KUKA KRL program: MyProgram_085().src

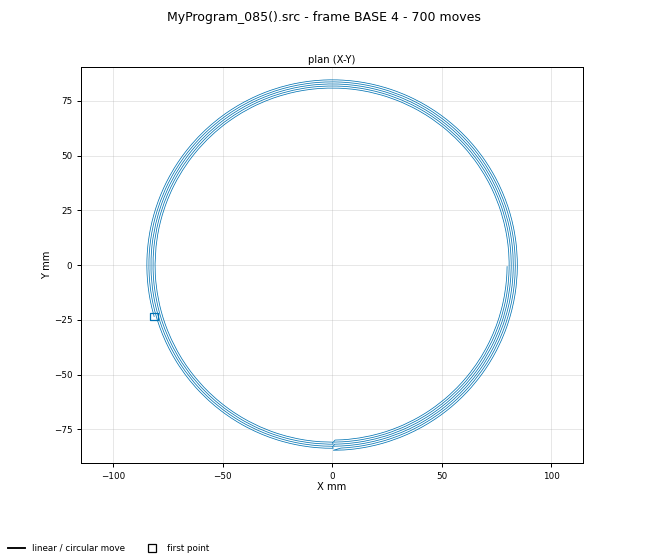
[picture p0: tool path of MyProgram_085().src in frame BASE 4, 700 of 700 moves have a stored position in this frame; points joined in program order, loops and branches not executed]
&ACCESS RVP
&REL 1
&PARAM TEMPLATE = C:\KRC\Roboter\Template\vorgabe
&PARAM EDITMASK = *
DEF MyProgram_085()
; ---- Setting reference (Base) ----
$BASE = BASE_DATA[4]

; --------------------------
; ---- Setting tool (TCP) ----
$TOOL = TOOL_DATA[3]
; --------------------------

$VEL.CP = VEL_APROX_PRINT
Startdeposition()
$VEL.CP = VEL_PRINT
LIN {X -81.258,Y -23.4932,Z 84,A -170.2717,B 24.9188,C -2.0806,E1 24.845,E2 255.2364} C_DIS
LIN {X -82.3528,Y -19.3072,Z 84,A -172.0172,B 24.9156,C -2.1214,E1 24.8439,E2 256.895} C_DIS
LIN {X -83.0894,Y -15.8383,Z 84,A -174.5177,B 24.9152,C -2.1261,E1 24.8425,E2 259.3989} C_DIS
LIN {X -83.5159,Y -13.4174,Z 84,A -176.5241,B 24.9155,C -2.122,E1 24.8416,E2 261.4269} C_DIS
LIN {X -83.9859,Y -10.0545,Z 84,A -178.7567,B 24.9148,C -2.1311,E1 24.8408,E2 263.6513} C_DIS
LIN {X -84.2675,Y -7.3389,Z 84,A 179.2872,B 24.9146,C -2.134,E1 24.8402,E2 265.6121} C_DIS
LIN {X -84.4963,Y -3.8886,Z 84,A 177.017,B 24.9138,C -2.1434,E1 24.8399,E2 267.8736} C_DIS
LIN {X -84.5836,Y -0.541,Z 84,A 174.7604,B 24.9132,C -2.1509,E1 24.8398,E2 270.1257} C_DIS
LIN {X -84.5494,Y 2.4664,Z 84,A 172.6653,B 24.9128,C -2.1559,E1 24.8399,E2 272.2217} C_DIS
LIN {X -84.435,Y 5.055,Z 84,A 170.8313,B 24.9125,C -2.1594,E1 24.8402,E2 274.0584} C_DIS
LIN {X -84.1499,Y 8.5742,Z 84,A 168.4952,B 24.9118,C -2.1685,E1 24.8408,E2 276.3867} C_DIS
LIN {X -83.8432,Y 11.1849,Z 84,A 166.6416,B 24.9115,C -2.1722,E1 24.8414,E2 278.2425} C_DIS
LIN {X -83.3207,Y 14.5775,Z 84,A 164.375,B 24.9108,C -2.1812,E1 24.8424,E2 280.5012} C_DIS
LIN {X -82.9257,Y 16.6767,Z 84,A 162.9181,B 24.9104,C -2.1855,E1 24.8432,E2 281.9565} C_DIS
LIN {X -82.2344,Y 19.8053,Z 84,A 160.6347,B 24.9101,C -2.1893,E1 24.8447,E2 284.2441} C_DIS
LIN {X -81.3682,Y 23.1062,Z 84,A 158.4682,B 24.9092,C -2.2004,E1 24.8463,E2 286.3966} C_DIS
LIN {X -80.4587,Y 26.0974,Z 84,A 156.0154,B 24.9094,C -2.198,E1 24.8483,E2 288.8692} C_DIS
LIN {X -79.338,Y 29.3307,Z 84,A 153.7423,B 24.9087,C -2.2063,E1 24.8505,E2 291.1354} C_DIS
LIN {X -78.306,Y 31.9821,Z 84,A 151.9175,B 24.908,C -2.2149,E1 24.8524,E2 292.9499} C_DIS
LIN {X -76.9778,Y 35.06,Z 84,A 149.7082,B 24.9073,C -2.2233,E1 24.8549,E2 295.1512} C_DIS
LIN {X -75.657,Y 37.8257,Z 84,A 147.6321,B 24.9068,C -2.2295,E1 24.8574,E2 297.2238} C_DIS
LIN {X -74.2269,Y 40.56,Z 84,A 145.2417,B 24.9069,C -2.2275,E1 24.8606,E2 299.6317} C_DIS
LIN {X -72.1363,Y 44.1714,Z 84,A 142.1378,B 24.9069,C -2.228,E1 24.8651,E2 302.7503} C_DIS
LIN {X -70.3586,Y 46.9528,Z 84,A 140.6207,B 24.9047,C -2.2536,E1 24.8673,E2 304.2139} C_DIS
LIN {X -68.1618,Y 50.0866,Z 84,A 137.8462,B 24.9045,C -2.2557,E1 24.8718,E2 306.997} C_DIS
LIN {X -66.2766,Y 52.5558,Z 84,A 135.0425,B 24.9057,C -2.2423,E1 24.8767,E2 309.8459} C_DIS
LIN {X -63.9412,Y 55.3742,Z 84,A 133.1912,B 24.9037,C -2.2657,E1 24.88,E2 311.6499} C_DIS
LIN {X -61.115,Y 58.4779,Z 84,A 130.1814,B 24.9035,C -2.2681,E1 24.8858,E2 314.667} C_DIS
LIN {X -58.0046,Y 61.5642,Z 84,A 127.0353,B 24.9033,C -2.2703,E1 24.8921,E2 317.8211} C_DIS
LIN {X -55.2393,Y 64.0587,Z 84,A 124.5405,B 24.9028,C -2.2767,E1 24.8973,E2 320.3105} C_DIS
LIN {X -51.7634,Y 66.8974,Z 84,A 121.7058,B 24.9017,C -2.2889,E1 24.9035,E2 323.1267} C_DIS
LIN {X -48.6455,Y 69.1989,Z 84,A 119.0158,B 24.9014,C -2.2924,E1 24.9096,E2 325.8177} C_DIS
LIN {X -46.1517,Y 70.8868,Z 84,A 116.9277,B 24.9012,C -2.2949,E1 24.9144,E2 327.9066} C_DIS
LIN {X -42.9543,Y 72.8671,Z 84,A 114.5021,B 24.9005,C -2.303,E1 24.9202,E2 330.3205} C_DIS
LIN {X -39.9938,Y 74.534,Z 84,A 111.9144,B 24.9008,C -2.2989,E1 24.9266,E2 332.9254} C_DIS
LIN {X -36.3147,Y 76.394,Z 84,A 109.3731,B 24.8999,C -2.3104,E1 24.9329,E2 335.4459} C_DIS
LIN {X -33.3203,Y 77.747,Z 84,A 107.1231,B 24.8996,C -2.3129,E1 24.9386,E2 337.6952} C_DIS
LIN {X -30.5085,Y 78.8929,Z 84,A 105.0579,B 24.8994,C -2.3155,E1 24.944,E2 339.7588} C_DIS
LIN {X -27.9226,Y 79.8437,Z 84,A 103.2111,B 24.8992,C -2.3184,E1 24.9489,E2 341.6024} C_DIS
LIN {X -23.5033,Y 81.2557,Z 84,A 99.7544,B 24.8996,C -2.3129,E1 24.9581,E2 345.0781} C_DIS
LIN {X -19.3603,Y 82.3405,Z 84,A 97.4785,B 24.8978,C -2.3338,E1 24.9642,E2 347.3076} C_DIS
LIN {X -17.0374,Y 82.8517,Z 84,A 95.5853,B 24.8984,C -2.3269,E1 24.9694,E2 349.2193} C_DIS
LIN {X -14.0779,Y 83.4057,Z 84,A 93.6062,B 24.8981,C -2.3302,E1 24.9748,E2 351.1926} C_DIS
LIN {X -10.9036,Y 83.8796,Z 84,A 91.394,B 24.8981,C -2.3305,E1 24.9809,E2 353.4059} C_DIS
LIN {X -7.5623,Y 84.2469,Z 84,A 88.9914,B 24.8983,C -2.328,E1 24.9876,E2 355.8159} C_DIS
LIN {X -3.933,Y 84.4944,Z 84,A 86.7832,B 24.8976,C -2.3365,E1 24.9937,E2 358.0046} C_DIS
LIN {X -1.2539,Y 84.5766,Z 84,A 84.7108,B 24.8982,C -2.3293,E1 24.9996,E2 360.0941} C_DIS
LIN {X 2.2908,Y 84.5548,Z 84,A 82.3368,B 24.8981,C -2.3305,E1 25.0062,E2 362.4651} C_DIS
LIN {X 4.9822,Y 84.439,Z 84,A 80.504,B 24.8981,C -2.3303,E1 25.0113,E2 364.2977} C_DIS
LIN {X 8.2772,Y 84.1808,Z 84,A 78.427,B 24.8977,C -2.3349,E1 25.017,E2 366.3625} C_DIS
LIN {X 11.0872,Y 83.8558,Z 84,A 76.403,B 24.898,C -2.3313,E1 25.0227,E2 368.3934} C_DIS
LIN {X 14.4147,Y 83.3494,Z 84,A 74.0384,B 24.8983,C -2.328,E1 25.0292,E2 370.7636} C_DIS
LIN {X 17.8759,Y 82.675,Z 84,A 71.6875,B 24.8983,C -2.3281,E1 25.0356,E2 373.1113} C_DIS
LIN {X 21.1707,Y 81.8932,Z 84,A 69.4403,B 24.8983,C -2.3282,E1 25.0417,E2 375.355} C_DIS
LIN {X 24.6364,Y 80.9192,Z 84,A 67.2437,B 24.8978,C -2.3339,E1 25.0476,E2 377.5343} C_DIS
LIN {X 26.9465,Y 80.1784,Z 84,A 65.4111,B 24.8984,C -2.3268,E1 25.0524,E2 379.3803} C_DIS
LIN {X 29.6504,Y 79.2189,Z 84,A 62.8102,B 24.9003,C -2.3047,E1 25.0594,E2 382.028} C_DIS
LIN {X 32.942,Y 77.9071,Z 84,A 61.3092,B 24.8981,C -2.3301,E1 25.0631,E2 383.4654} C_DIS
LIN {X 35.0479,Y 76.9832,Z 84,A 59.6938,B 24.8984,C -2.3265,E1 25.0672,E2 385.0853} C_DIS
LIN {X 37.4119,Y 75.862,Z 84,A 57.6987,B 24.8992,C -2.3174,E1 25.0723,E2 387.0968} C_DIS
LIN {X 40.5488,Y 74.2329,Z 84,A 55.247,B 24.8997,C -2.3124,E1 25.0783,E2 389.5533} C_DIS
LIN {X 43.6284,Y 72.4663,Z 84,A 52.8273,B 24.9,C -2.3085,E1 25.0842,E2 391.9749} C_DIS
LIN {X 46.9407,Y 70.3665,Z 84,A 50.2167,B 24.9003,C -2.3058,E1 25.0903,E2 394.5835} C_DIS
LIN {X 49.6746,Y 68.4634,Z 84,A 48.0134,B 24.9004,C -2.3037,E1 25.0953,E2 396.7841} C_DIS
LIN {X 52.2744,Y 66.4989,Z 84,A 45.8438,B 24.9007,C -2.3009,E1 25.1001,E2 398.9522} C_DIS
LIN {X 54.843,Y 64.3966,Z 84,A 43.7202,B 24.9007,C -2.3007,E1 25.1046,E2 401.0682} C_DIS
LIN {X 56.9564,Y 62.5359,Z 84,A 41.8463,B 24.9009,C -2.298,E1 25.1085,E2 402.941} C_DIS
LIN {X 59.0852,Y 60.5299,Z 84,A 39.6486,B 24.9019,C -2.2869,E1 25.113,E2 405.1558} C_DIS
LIN {X 61.4852,Y 58.0886,Z 84,A 37.4909,B 24.9019,C -2.2871,E1 25.1172,E2 407.3036} C_DIS
LIN {X 64.1932,Y 55.0818,Z 84,A 34.6835,B 24.9026,C -2.2788,E1 25.1224,E2 410.1182} C_DIS
LIN {X 66.2537,Y 52.5847,Z 84,A 32.5055,B 24.903,C -2.2741,E1 25.1262,E2 412.2971} C_DIS
LIN {X 68.4835,Y 49.6473,Z 84,A 30.195,B 24.903,C -2.2741,E1 25.13,E2 414.5964} C_DIS
LIN {X 70.0955,Y 47.3425,Z 84,A 28.0798,B 24.904,C -2.2625,E1 25.1334,E2 416.7288} C_DIS
LIN {X 71.8637,Y 44.6132,Z 84,A 25.9695,B 24.9042,C -2.2599,E1 25.1366,E2 418.8348} C_DIS
LIN {X 73.3555,Y 42.1147,Z 84,A 24.0489,B 24.9045,C -2.2563,E1 25.1393,E2 420.7539} C_DIS
LIN {X 74.5437,Y 39.976,Z 84,A 22.2403,B 24.9053,C -2.2468,E1 25.1417,E2 422.5754} C_DIS
LIN {X 76.1666,Y 36.7879,Z 84,A 19.9576,B 24.9055,C -2.2448,E1 25.1445,E2 424.8508} C_DIS
LIN {X 77.7532,Y 33.3037,Z 84,A 16.6318,B 24.9081,C -2.2133,E1 25.1483,E2 428.2328} C_DIS
LIN {X 79.201,Y 29.6977,Z 84,A 14.5929,B 24.9071,C -2.2252,E1 25.1503,E2 430.2322} C_DIS
LIN {X 80.3308,Y 26.4926,Z 84,A 12.4263,B 24.9073,C -2.2228,E1 25.1522,E2 432.3922} C_DIS
LIN {X 81.2016,Y 23.6879,Z 84,A 10.4534,B 24.9078,C -2.2174,E1 25.1538,E2 434.3665} C_DIS
LIN {X 82.0478,Y 20.569,Z 84,A 8.2194,B 24.9084,C -2.2093,E1 25.1554,E2 436.6069} C_DIS
LIN {X 82.8109,Y 17.2361,Z 84,A 5.9479,B 24.9089,C -2.2037,E1 25.1568,E2 438.8784} C_DIS
LIN {X 83.338,Y 14.4812,Z 84,A 4.0007,B 24.9095,C -2.1962,E1 25.1577,E2 440.832} C_DIS
LIN {X 83.8789,Y 10.9088,Z 84,A 1.8383,B 24.9094,C -2.1981,E1 25.1586,E2 442.9771} C_DIS
LIN {X 84.2078,Y 7.9856,Z 84,A -0.6462,B 24.9112,C -2.1753,E1 25.1593,E2 445.5006} C_DIS
LIN {X 84.5468,Y 2.554,Z 84,A -4.3801,B 24.9123,C -2.162,E1 25.1598,E2 449.2437} C_DIS
LIN {X 84.5806,Y -1.0264,Z 84,A -6.4606,B 24.912,C -2.1658,E1 25.1598,E2 451.303} C_DIS
LIN {X 84.4797,Y -4.247,Z 84,A -8.5268,B 24.9123,C -2.1627,E1 25.1595,E2 453.3642} C_DIS
LIN {X 83.9739,Y -10.1565,Z 84,A -12.6253,B 24.9135,C -2.1471,E1 25.1584,E2 457.4751} C_DIS
LIN {X 83.5288,Y -13.3334,Z 84,A -15.2054,B 24.9152,C -2.1266,E1 25.1573,E2 460.0886} C_DIS
LIN {X 82.9598,Y -16.5061,Z 84,A -17.3336,B 24.9156,C -2.1215,E1 25.1561,E2 462.2163} C_DIS
LIN {X 82.0892,Y -20.4002,Z 84,A -19.606,B 24.9151,C -2.1273,E1 25.1547,E2 464.4618} C_DIS
LIN {X 81.2074,Y -23.6685,Z 84,A -21.9819,B 24.9159,C -2.1174,E1 25.1529,E2 466.8476} C_DIS
LIN {X 80.088,Y -27.2145,Z 84,A -24.189,B 24.9157,C -2.12,E1 25.151,E2 469.0359} C_DIS
LIN {X 78.9874,Y -30.2617,Z 84,A -26.4098,B 24.9163,C -2.1124,E1 25.1488,E2 471.2624} C_DIS
LIN {X 77.352,Y -34.2281,Z 84,A -30.4851,B 24.9201,C -2.0648,E1 25.1442,E2 475.4278} C_DIS
LIN {X 75.1596,Y -38.8052,Z 84,A -32.3854,B 24.9168,C -2.1057,E1 25.142,E2 477.2213} C_DIS
LIN {X 73.4267,Y -41.9908,Z 84,A -35.7576,B 24.9198,C -2.068,E1 25.1373,E2 480.6649} C_DIS
LIN {X 71.7723,Y -44.7595,Z 84,A -37.2898,B 24.9186,C -2.0835,E1 25.1351,E2 482.1527} C_DIS
LIN {X 70.1825,Y -47.214,Z 84,A -39.3837,B 24.9193,C -2.0742,E1 25.1319,E2 484.2582} C_DIS
LIN {X 68.3451,Y -49.8363,Z 84,A -41.5585,B 24.9198,C -2.0681,E1 25.1283,E2 486.4368} C_DIS
LIN {X 66.5336,Y -52.2306,Z 84,A -43.9673,B 24.9212,C -2.0503,E1 25.1242,E2 488.8764} C_DIS
LIN {X 63.5973,Y -55.7682,Z 84,A -46.5786,B 24.9205,C -2.0589,E1 25.1195,E2 491.4554} C_DIS
LIN {X 61.6049,Y -57.9613,Z 84,A -48.5956,B 24.9209,C -2.0535,E1 25.1157,E2 493.4762} C_DIS
LIN {X 59.4587,Y -60.161,Z 84,A -50.6632,B 24.9213,C -2.0489,E1 25.1116,E2 495.546} C_DIS
LIN {X 57.2741,Y -62.2444,Z 84,A -52.8275,B 24.9219,C -2.0402,E1 25.1072,E2 497.722} C_DIS
LIN {X 54.4849,Y -64.7017,Z 84,A -55.2672,B 24.9222,C -2.037,E1 25.102,E2 500.1595} C_DIS
LIN {X 52.1024,Y -66.6349,Z 84,A -57.3582,B 24.9226,C -2.0321,E1 25.0974,E2 502.2544} C_DIS
LIN {X 49.6131,Y -68.5085,Z 84,A -59.3441,B 24.9226,C -2.0318,E1 25.093,E2 504.234} C_DIS
LIN {X 46.7155,Y -70.5151,Z 84,A -61.7837,B 24.9231,C -2.0254,E1 25.0873,E2 506.6805} C_DIS
LIN {X 44.0739,Y -72.1955,Z 84,A -63.9286,B 24.9234,C -2.0206,E1 25.0822,E2 508.8298} C_DIS
LIN {X 40.9406,Y -74.0179,Z 84,A -67.0141,B 24.9253,C -1.996,E1 25.0746,E2 511.9643} C_DIS
LIN {X 37.734,Y -75.7024,Z 84,A -68.9066,B 24.9243,C -2.0099,E1 25.07,E2 513.8188} C_DIS
LIN {X 34.381,Y -77.2838,Z 84,A -71.9632,B 24.9258,C -1.9887,E1 25.0621,E2 516.9181} C_DIS
LIN {X 31.0532,Y -78.6791,Z 84,A -73.3423,B 24.9236,C -2.0192,E1 25.0587,E2 518.2219} C_DIS
LIN {X 25.9181,Y -80.5167,Z 84,A -77.3653,B 24.9247,C -2.0039,E1 25.0481,E2 522.2728} C_DIS
LIN {X 23.0747,Y -81.3771,Z 84,A -79.3426,B 24.9247,C -2.0028,E1 25.0428,E2 524.2494} C_DIS
LIN {X 20.0403,Y -82.177,Z 84,A -81.8961,B 24.926,C -1.9872,E1 25.0358,E2 526.836} C_DIS
LIN {X 16.4441,Y -82.9728,Z 84,A -83.8435,B 24.9248,C -2.0021,E1 25.0306,E2 528.7456} C_DIS
LIN {X 13.908,Y -83.4341,Z 84,A -85.8616,B 24.9256,C -1.9923,E1 25.0249,E2 530.7849} C_DIS
LIN {X 10.3473,Y -83.9514,Z 84,A -88.0451,B 24.9251,C -1.9985,E1 25.0189,E2 532.9517} C_DIS
LIN {X 7.3763,Y -84.264,Z 84,A -90.0792,B 24.9252,C -1.9971,E1 25.0133,E2 534.9878} C_DIS
LIN {X 5.3469,Y -84.4169,Z 84,A -91.6987,B 24.9258,C -1.989,E1 25.0087,E2 536.6258} C_DIS
LIN {X 0.5554,Y -84.5445,Z 84,A -94.0902,B 24.9239,C -2.0151,E1 25.0023,E2 538.9549} C_DIS
Enddeposition()
LIN {X 0.5554,Y -84.5445,Z 84,A -94.0902,B 24.9239,C -2.0151,E1 25.0023,E2 538.9549} C_DIS
Startdeposition()
$VEL.CP = VEL_PRINT
LIN {X 4.0199,Y -83.5536,Z 84,A -91.4821,B 24.9221,C -2.0387,E1 25.0097,E2 536.2916} C_DIS
LIN {X 7.177,Y -83.3423,Z 84,A -88.8971,B 24.921,C -2.0528,E1 25.0169,E2 533.6745} C_DIS
LIN {X 11.2811,Y -82.8861,Z 84,A -86.5387,B 24.922,C -2.0398,E1 25.0234,E2 531.3487} C_DIS
LIN {X 14.1672,Y -82.4416,Z 84,A -84.4181,B 24.9216,C -2.0451,E1 25.0293,E2 529.2177} C_DIS
LIN {X 18.2064,Y -81.6443,Z 84,A -81.4549,B 24.921,C -2.0521,E1 25.0374,E2 526.2417} C_DIS
LIN {X 23.7052,Y -80.22,Z 84,A -77.9146,B 24.9216,C -2.0451,E1 25.0469,E2 522.7236} C_DIS
LIN {X 26.3192,Y -79.4006,Z 84,A -75.1328,B 24.9191,C -2.0764,E1 25.0544,E2 519.8729} C_DIS
LIN {X 30.3174,Y -77.9623,Z 84,A -73.2321,B 24.9214,C -2.0478,E1 25.0592,E2 518.0441} C_DIS
LIN {X 34.0465,Y -76.4077,Z 84,A -70.3229,B 24.9207,C -2.0564,E1 25.0667,E2 515.1215} C_DIS
LIN {X 35.9853,Y -75.5137,Z 84,A -68.6164,B 24.9199,C -2.0666,E1 25.0711,E2 513.3953} C_DIS
LIN {X 40.6616,Y -73.1016,Z 84,A -65.0227,B 24.9195,C -2.0724,E1 25.0799,E2 509.7981} C_DIS
LIN {X 45.2214,Y -70.3719,Z 84,A -60.7698,B 24.9173,C -2.0994,E1 25.0901,E2 505.4948} C_DIS
LIN {X 48.8035,Y -67.9373,Z 84,A -58.3698,B 24.9183,C -2.0867,E1 25.0955,E2 503.1333} C_DIS
LIN {X 52.051,Y -65.4823,Z 84,A -55.9631,B 24.9189,C -2.0801,E1 25.1007,E2 500.7511} C_DIS
LIN {X 54.2015,Y -63.7133,Z 84,A -54.2455,B 24.919,C -2.0781,E1 25.1044,E2 499.0447} C_DIS
LIN {X 57.1138,Y -61.1168,Z 84,A -50.9148,B 24.9168,C -2.1061,E1 25.1114,E2 495.6614} C_DIS
LIN {X 60.324,Y -57.9501,Z 84,A -48.2074,B 24.9172,C -2.1009,E1 25.1166,E2 492.9778} C_DIS
LIN {X 62.4733,Y -55.6266,Z 84,A -45.5471,B 24.9155,C -2.1228,E1 25.1217,E2 490.2776} C_DIS
LIN {X 64.6916,Y -53.031,Z 84,A -43.7656,B 24.9165,C -2.1102,E1 25.1248,E2 488.534} C_DIS
LIN {X 68.6131,Y -47.8481,Z 84,A -38.7416,B 24.914,C -2.1415,E1 25.1331,E2 483.4604} C_DIS
LIN {X 70.6127,Y -44.8463,Z 84,A -36.3085,B 24.9135,C -2.1472,E1 25.1368,E2 481.0261} C_DIS
LIN {X 72.409,Y -41.8828,Z 84,A -34.6666,B 24.915,C -2.1293,E1 25.139,E2 479.4348} C_DIS
LIN {X 74.0802,Y -38.8501,Z 84,A -32.4822,B 24.915,C -2.1299,E1 25.1419,E2 477.2604} C_DIS
LIN {X 76.2889,Y -34.3102,Z 84,A -28.9902,B 24.914,C -2.1413,E1 25.1462,E2 473.7603} C_DIS
LIN {X 77.8847,Y -30.515,Z 84,A -25.8854,B 24.9125,C -2.1594,E1 25.1495,E2 470.6298} C_DIS
LIN {X 79.1087,Y -27.1888,Z 84,A -22.8184,B 24.9101,C -2.1886,E1 25.1523,E2 467.5111} C_DIS
LIN {X 80.2758,Y -23.5171,Z 84,A -20.9909,B 24.9117,C -2.1693,E1 25.1538,E2 465.7397} C_DIS
LIN {X 81.0511,Y -20.6864,Z 84,A -19.0499,B 24.9114,C -2.1733,E1 25.1551,E2 463.8005} C_DIS
LIN {X 81.9401,Y -16.8226,Z 84,A -15.9084,B 24.9095,C -2.1963,E1 25.157,E2 460.6229} C_DIS
LIN {X 82.6235,Y -13.0619,Z 84,A -13.2409,B 24.9087,C -2.2063,E1 25.1582,E2 457.9474} C_DIS
LIN {X 83.0754,Y -9.7807,Z 84,A -10.9669,B 24.9081,C -2.2137,E1 25.159,E2 455.6693} C_DIS
LIN {X 83.4824,Y -5.2907,Z 84,A -7.8895,B 24.9073,C -2.2232,E1 25.1596,E2 452.5877} C_DIS
LIN {X 83.6471,Y -0.6032,Z 84,A -3.9008,B 24.9042,C -2.2601,E1 25.1597,E2 448.5358} C_DIS
LIN {X 83.5087,Y 4.8515,Z 84,A -1.6888,B 24.9076,C -2.22,E1 25.1595,E2 446.4316} C_DIS
LIN {X 83.3102,Y 7.5248,Z 84,A 0.3928,B 24.9064,C -2.2341,E1 25.159,E2 444.3291} C_DIS
LIN {X 82.9542,Y 10.7605,Z 84,A 2.5084,B 24.9061,C -2.2372,E1 25.1583,E2 442.2185} C_DIS
LIN {X 82.5337,Y 13.6166,Z 84,A 4.5625,B 24.9054,C -2.246,E1 25.1574,E2 440.1558} C_DIS
LIN {X 81.966,Y 16.6967,Z 84,A 6.6673,B 24.9049,C -2.2513,E1 25.1563,E2 438.0509} C_DIS
LIN {X 81.2888,Y 19.7312,Z 84,A 8.4277,B 24.9054,C -2.2454,E1 25.1552,E2 436.3145} C_DIS
LIN {X 80.2379,Y 23.6451,Z 84,A 11.5985,B 24.9036,C -2.267,E1 25.1529,E2 433.111} C_DIS
LIN {X 79.2298,Y 26.8297,Z 84,A 14.4891,B 24.9013,C -2.294,E1 25.1502,E2 430.1728} C_DIS
LIN {X 78.0075,Y 30.202,Z 84,A 16.0399,B 24.9033,C -2.2708,E1 25.1488,E2 428.6856} C_DIS
LIN {X 76.2468,Y 34.4035,Z 84,A 19.2998,B 24.9021,C -2.2843,E1 25.1452,E2 425.4115} C_DIS
LIN {X 75.0446,Y 36.9533,Z 84,A 21.295,B 24.9015,C -2.2918,E1 25.1428,E2 423.4093} C_DIS
LIN {X 73.6627,Y 39.6367,Z 84,A 23.3793,B 24.9009,C -2.298,E1 25.14,E2 421.3214} C_DIS
LIN {X 72.552,Y 41.634,Z 84,A 25.2545,B 24.8997,C -2.3125,E1 25.1374,E2 419.4218} C_DIS
LIN {X 70.2759,Y 45.3709,Z 84,A 27.7115,B 24.9005,C -2.3024,E1 25.1338,E2 417.001} C_DIS
LIN {X 68.4525,Y 48.0791,Z 84,A 30.096,B 24.8996,C -2.3129,E1 25.13,E2 414.6035} C_DIS
LIN {X 66.2527,Y 51.0663,Z 84,A 32.5388,B 24.8994,C -2.3159,E1 25.126,E2 412.1654} C_DIS
LIN {X 64.7282,Y 52.9868,Z 84,A 34.348,B 24.8987,C -2.324,E1 25.1228,E2 410.3453} C_DIS
LIN {X 62.2646,Y 55.8597,Z 84,A 37.2769,B 24.8972,C -2.3409,E1 25.1173,E2 407.3895} C_DIS
LIN {X 59.4362,Y 58.8603,Z 84,A 39.6235,B 24.898,C -2.3314,E1 25.1128,E2 405.0755} C_DIS
LIN {X 57.3676,Y 60.8781,Z 84,A 41.4708,B 24.898,C -2.3313,E1 25.1091,E2 403.2362} C_DIS
LIN {X 54.5044,Y 63.4552,Z 84,A 44.3183,B 24.897,C -2.3432,E1 25.1031,E2 400.372} C_DIS
LIN {X 51.9825,Y 65.5364,Z 84,A 46.598,B 24.8965,C -2.3486,E1 25.0982,E2 398.088} C_DIS
LIN {X 50.1123,Y 66.9773,Z 84,A 48.6395,B 24.895,C -2.3651,E1 25.0936,E2 396.0147} C_DIS
LIN {X 46.3142,Y 69.6583,Z 84,A 51.7223,B 24.8949,C -2.367,E1 25.0864,E2 392.9379} C_DIS
LIN {X 43.1556,Y 71.6582,Z 84,A 54.0955,B 24.8951,C -2.3648,E1 25.0808,E2 390.5773} C_DIS
LIN {X 39.9157,Y 73.5113,Z 84,A 56.3672,B 24.8956,C -2.3593,E1 25.0753,E2 388.3253} C_DIS
LIN {X 37.3694,Y 74.8383,Z 84,A 58.3963,B 24.8952,C -2.3638,E1 25.0703,E2 386.2912} C_DIS
LIN {X 35.4416,Y 75.77,Z 84,A 60.1955,B 24.8941,C -2.376,E1 25.0657,E2 384.4676} C_DIS
LIN {X 32.1295,Y 77.2336,Z 84,A 62.6353,B 24.8939,C -2.3773,E1 25.0594,E2 382.0305} C_DIS
LIN {X 25.6498,Y 79.6196,Z 84,A 66.7451,B 24.8953,C -2.3622,E1 25.0487,E2 377.9649} C_DIS
LIN {X 21.7213,Y 80.7798,Z 84,A 69.8965,B 24.8942,C -2.3748,E1 25.0402,E2 374.7891} C_DIS
LIN {X 19.5659,Y 81.3291,Z 84,A 71.4985,B 24.8939,C -2.378,E1 25.0358,E2 373.1816} C_DIS
LIN {X 16.3067,Y 82.0459,Z 84,A 73.6895,B 24.8941,C -2.3761,E1 25.0298,E2 370.9979} C_DIS
LIN {X 13.4669,Y 82.5587,Z 84,A 75.5595,B 24.8943,C -2.3736,E1 25.0247,E2 369.1358} C_DIS
LIN {X 10.6013,Y 82.9748,Z 84,A 77.7465,B 24.8937,C -2.3803,E1 25.0186,E2 366.9349} C_DIS
LIN {X 6.8638,Y 83.3673,Z 84,A 80.1558,B 24.8941,C -2.3755,E1 25.012,E2 364.5383} C_DIS
LIN {X 4.0104,Y 83.554,Z 84,A 82.163,B 24.894,C -2.3769,E1 25.0064,E2 362.5285} C_DIS
LIN {X 0.8514,Y 83.6455,Z 84,A 84.5138,B 24.8935,C -2.3822,E1 24.9998,E2 360.1655} C_DIS
LIN {X -3.0959,Y 83.5933,Z 84,A 87.0781,B 24.8939,C -2.3773,E1 24.9926,E2 357.6125} C_DIS
LIN {X -6.2001,Y 83.4204,Z 84,A 89.1931,B 24.8941,C -2.376,E1 24.9868,E2 355.4999} C_DIS
LIN {X -9.1905,Y 83.1442,Z 84,A 91.038,B 24.8947,C -2.3687,E1 24.9817,E2 353.6714} C_DIS
LIN {X -11.4027,Y 82.8691,Z 84,A 93.1008,B 24.8934,C -2.3836,E1 24.9759,E2 351.5716} C_DIS
LIN {X -15.7052,Y 82.1617,Z 84,A 95.754,B 24.8945,C -2.3715,E1 24.9686,E2 348.9444} C_DIS
LIN {X -19.0218,Y 81.4579,Z 84,A 98.6644,B 24.8931,C -2.3867,E1 24.9606,E2 345.9941} C_DIS
LIN {X -22.388,Y 80.5987,Z 84,A 100.5352,B 24.8947,C -2.3693,E1 24.9557,E2 344.1617} C_DIS
LIN {X -26.2545,Y 79.4231,Z 84,A 103.3416,B 24.8948,C -2.3673,E1 24.9482,E2 341.3552} C_DIS
LIN {X -30.6618,Y 77.827,Z 84,A 106.4606,B 24.8954,C -2.3605,E1 24.9401,E2 338.246} C_DIS
LIN {X -33.92,Y 76.4642,Z 84,A 108.7711,B 24.896,C -2.3539,E1 24.9342,E2 335.9457} C_DIS
LIN {X -36.6181,Y 75.2096,Z 84,A 110.7014,B 24.8966,C -2.3477,E1 24.9293,E2 334.0254} C_DIS
LIN {X -41.6829,Y 72.5239,Z 84,A 114.355,B 24.8978,C -2.3333,E1 24.9204,E2 330.3957} C_DIS
LIN {X -45.6654,Y 70.0861,Z 84,A 117.8635,B 24.8976,C -2.3361,E1 24.912,E2 326.8697} C_DIS
LIN {X -48.5182,Y 68.1409,Z 84,A 119.9993,B 24.8986,C -2.325,E1 24.9071,E2 324.753} C_DIS
LIN {X -51.0495,Y 66.2656,Z 84,A 123.1178,B 24.8966,C -2.3474,E1 24.9,E2 321.5699} C_DIS
LIN {X -55.1202,Y 62.9203,Z 84,A 126.24,B 24.8985,C -2.3258,E1 24.8935,E2 318.4872} C_DIS
LIN {X -57.718,Y 60.5474,Z 84,A 128.745,B 24.8988,C -2.3229,E1 24.8883,E2 315.979} C_DIS
LIN {X -60.148,Y 58.1327,Z 84,A 131.1062,B 24.8992,C -2.3176,E1 24.8837,E2 313.6202} C_DIS
LIN {X -62.7845,Y 55.2757,Z 84,A 133.9449,B 24.8994,C -2.3158,E1 24.8784,E2 310.7731} C_DIS
LIN {X -65.7821,Y 51.6717,Z 84,A 136.9232,B 24.9007,C -2.3011,E1 24.8732,E2 307.8162} C_DIS
LIN {X -67.6029,Y 49.2652,Z 84,A 139.4161,B 24.9001,C -2.3072,E1 24.869,E2 305.2965} C_DIS
LIN {X -69.6073,Y 46.3916,Z 84,A 142.338,B 24.8994,C -2.315,E1 24.8645,E2 302.3414} C_DIS
LIN {X -71.9297,Y 42.7004,Z 84,A 144.0334,B 24.9032,C -2.2712,E1 24.8622,E2 300.742} C_DIS
LIN {X -72.8535,Y 41.1046,Z 84,A 145.9824,B 24.9019,C -2.2862,E1 24.8594,E2 298.747} C_DIS
LIN {X -74.8442,Y 37.3574,Z 84,A 148.6191,B 24.9033,C -2.2703,E1 24.856,E2 296.134} C_DIS
LIN {X -76.1404,Y 34.6397,Z 84,A 150.7736,B 24.9036,C -2.2667,E1 24.8535,E2 293.9764} C_DIS
LIN {X -78.4276,Y 29.0948,Z 84,A 154.6871,B 24.9051,C -2.2489,E1 24.8495,E2 290.0835} C_DIS
LIN {X -80.0105,Y 24.406,Z 84,A 158.3357,B 24.9054,C -2.2454,E1 24.8463,E2 286.4224} C_DIS
LIN {X -80.8652,Y 21.405,Z 84,A 160.4607,B 24.906,C -2.2384,E1 24.8447,E2 284.3019} C_DIS
LIN {X -81.6261,Y 18.2919,Z 84,A 162.4236,B 24.9071,C -2.2252,E1 24.8435,E2 282.3589} C_DIS
LIN {X -82.3773,Y 14.5338,Z 84,A 165.282,B 24.9073,C -2.2232,E1 24.842,E2 279.4884} C_DIS
LIN {X -82.853,Y 11.5161,Z 84,A 167.3007,B 24.908,C -2.2145,E1 24.8411,E2 277.4784} C_DIS
LIN {X -83.2566,Y 8.1054,Z 84,A 169.7488,B 24.9084,C -2.2096,E1 24.8404,E2 275.0274} C_DIS
LIN {X -83.486,Y 5.2374,Z 84,A 171.8714,B 24.9086,C -2.2074,E1 24.84,E2 272.8973} C_DIS
LIN {X -83.6086,Y 2.6043,Z 84,A 173.8259,B 24.9087,C -2.2057,E1 24.8398,E2 270.935} C_DIS
LIN {X -83.6345,Y -1.5646,Z 84,A 176.4351,B 24.91,C -2.1899,E1 24.8398,E2 268.3478} C_DIS
LIN {X -83.5095,Y -4.8361,Z 84,A 178.371,B 24.9113,C -2.1746,E1 24.8401,E2 266.437} C_DIS
LIN {X -83.3214,Y -7.4037,Z 84,A -179.3843,B 24.9107,C -2.182,E1 24.8406,E2 264.1611} C_DIS
LIN {X -82.8773,Y -11.3456,Z 84,A -176.7111,B 24.9115,C -2.1722,E1 24.8415,E2 261.4951} C_DIS
LIN {X -82.3288,Y -14.8035,Z 84,A -173.8613,B 24.9111,C -2.1771,E1 24.8429,E2 258.6167} C_DIS
LIN {X -81.697,Y -17.9666,Z 84,A -172.3552,B 24.9132,C -2.1512,E1 24.8438,E2 257.1637} C_DIS
LIN {X -80.9704,Y -20.9996,Z 84,A -169.6186,B 24.9124,C -2.1611,E1 24.8457,E2 254.3876} C_DIS
LIN {X -79.8108,Y -25.0499,Z 84,A -166.9227,B 24.9135,C -2.1472,E1 24.8478,E2 251.7091} C_DIS
LIN {X -78.5877,Y -28.6558,Z 84,A -164.5467,B 24.9147,C -2.1332,E1 24.85,E2 249.3531} C_DIS
LIN {X -77.4142,Y -31.6899,Z 84,A -162.5688,B 24.9157,C -2.1199,E1 24.852,E2 247.3958} C_DIS
LIN {X -75.9889,Y -34.9715,Z 84,A -159.701,B 24.9154,C -2.1244,E1 24.8553,E2 244.5016} C_DIS
LIN {X -74.3359,Y -38.3596,Z 84,A -157.4418,B 24.9166,C -2.1084,E1 24.8581,E2 242.2683} C_DIS
LIN {X -72.555,Y -41.6288,Z 84,A -154.6621,B 24.9166,C -2.1079,E1 24.8618,E2 239.4752} C_DIS
LIN {X -70.9838,Y -44.2549,Z 84,A -152.5009,B 24.917,C -2.1042,E1 24.865,E2 237.3117} C_DIS
LIN {X -69.7977,Y -46.1028,Z 84,A -150.0116,B 24.9151,C -2.1281,E1 24.869,E2 234.7531} C_DIS
LIN {X -67.1241,Y -49.9169,Z 84,A -147.7577,B 24.9178,C -2.0939,E1 24.8726,E2 232.5699} C_DIS
LIN {X -64.8222,Y -52.8709,Z 84,A -144.4317,B 24.9166,C -2.1093,E1 24.8785,E2 229.1914} C_DIS
LIN {X -62.2432,Y -55.8837,Z 84,A -142.6032,B 24.919,C -2.0781,E1 24.8817,E2 227.4292} C_DIS
LIN {X -60.5307,Y -57.7357,Z 84,A -140.6584,B 24.9188,C -2.0805,E1 24.8855,E2 225.4704} C_DIS
LIN {X -56.3991,Y -61.7768,Z 84,A -136.6948,B 24.9195,C -2.0725,E1 24.8935,E2 221.5093} C_DIS
LIN {X -53.6227,Y -64.2015,Z 84,A -133.558,B 24.9185,C -2.0853,E1 24.9003,E2 218.3299} C_DIS
LIN {X -50.7457,Y -66.4997,Z 84,A -131.6469,B 24.9202,C -2.0632,E1 24.9044,E2 216.4645} C_DIS
LIN {X -48.781,Y -67.9533,Z 84,A -129.4774,B 24.9193,C -2.0747,E1 24.9094,E2 214.2599} C_DIS
LIN {X -46.1249,Y -69.7831,Z 84,A -127.6266,B 24.9204,C -2.0608,E1 24.9136,E2 212.4362} C_DIS
LIN {X -43.2256,Y -71.6156,Z 84,A -125.5331,B 24.9212,C -2.0499,E1 24.9186,E2 210.3621} C_DIS
LIN {X -40.8323,Y -73.0062,Z 84,A -123.6268,B 24.9214,C -2.0476,E1 24.9232,E2 208.4558} C_DIS
LIN {X -39.0883,Y -73.9547,Z 84,A -121.8503,B 24.9206,C -2.058,E1 24.9276,E2 206.6494} C_DIS
LIN {X -35.2729,Y -75.8486,Z 84,A -118.6111,B 24.9201,C -2.0642,E1 24.9359,E2 203.3875} C_DIS
LIN {X -31.9626,Y -77.3032,Z 84,A -116.1232,B 24.9203,C -2.062,E1 24.9423,E2 200.8992} C_DIS
LIN {X -28.6867,Y -78.5764,Z 84,A -114.6751,B 24.9226,C -2.0313,E1 24.9459,E2 199.521} C_DIS
LIN {X -24.7899,Y -79.8915,Z 84,A -111.5118,B 24.922,C -2.0393,E1 24.9544,E2 196.3327} C_DIS
LIN {X -22.6359,Y -80.5284,Z 84,A -109.8927,B 24.922,C -2.0407,E1 24.9587,E2 194.7077} C_DIS
LIN {X -19.4479,Y -81.3579,Z 84,A -107.7206,B 24.9222,C -2.037,E1 24.9646,E2 192.5415} C_DIS
LIN {X -16.5834,Y -81.9892,Z 84,A -105.7636,B 24.9224,C -2.0345,E1 24.9699,E2 190.5879} C_DIS
LIN {X -13.726,Y -82.5154,Z 84,A -103.6716,B 24.9222,C -2.037,E1 24.9757,E2 188.4881} C_DIS
LIN {X -10.1382,Y -83.0334,Z 84,A -101.2301,B 24.9223,C -2.0352,E1 24.9824,E2 186.0489} C_DIS
LIN {X -7.1797,Y -83.342,Z 84,A -98.4247,B 24.9205,C -2.0588,E1 24.9904,E2 183.1863} C_DIS
LIN {X -3.1986,Y -83.5889,Z 84,A -96.4065,B 24.9222,C -2.0369,E1 24.9959,E2 181.2195} C_DIS
LIN {X -0.9118,Y -83.6451,Z 84,A -94.9838,B 24.9225,C -2.0327,E1 24.9998,E2 179.8066} C_DIS
LIN {X 0.5326,Y -83.6418,Z 84,A -93.41,B 24.9211,C -2.0512,E1 25.0044,E2 178.1891} C_DIS
Enddeposition()
LIN {X 0.5326,Y -83.6418,Z 84,A -93.41,B 24.9211,C -2.0512,E1 25.0044,E2 178.1891} C_DIS
Startdeposition()
$VEL.CP = VEL_PRINT
LIN {X 0.1012,Y -82.7139,Z 84,A -95.3168,B 24.9236,C -2.0181,E1 24.9988,E2 180.1743} C_DIS
LIN {X -3.8669,Y -82.6232,Z 84,A -98.524,B 24.9247,C -2.0043,E1 24.9898,E2 183.4149} C_DIS
LIN {X -7.069,Y -82.4118,Z 84,A -100.038,B 24.9231,C -2.0253,E1 24.9857,E2 184.8798} C_DIS
LIN {X -9.4478,Y -82.1718,Z 84,A -101.8874,B 24.9235,C -2.0197,E1 24.9805,E2 186.7434} C_DIS
LIN {X -13.2784,Y -81.641,Z 84,A -104.7676,B 24.9239,C -2.0145,E1 24.9725,E2 189.6385} C_DIS
LIN {X -16.5328,Y -81.0439,Z 84,A -106.8623,B 24.9234,C -2.0211,E1 24.9668,E2 191.7198} C_DIS
LIN {X -19.8829,Y -80.2882,Z 84,A -109.6271,B 24.9242,C -2.0112,E1 24.9592,E2 194.512} C_DIS
LIN {X -23.4792,Y -79.3106,Z 84,A -112.0863,B 24.9238,C -2.0164,E1 24.9527,E2 196.9627} C_DIS
LIN {X -27.1139,Y -78.1432,Z 84,A -114.4881,B 24.9231,C -2.0255,E1 24.9463,E2 199.3475} C_DIS
LIN {X -30.9706,Y -76.6963,Z 84,A -118.0113,B 24.9243,C -2.0091,E1 24.9371,E2 202.9171} C_DIS
LIN {X -34.3495,Y -75.2444,Z 84,A -119.6361,B 24.9221,C -2.0381,E1 24.9331,E2 204.477} C_DIS
LIN {X -39.3816,Y -72.7361,Z 84,A -123.5942,B 24.9219,C -2.0411,E1 24.9232,E2 208.4385} C_DIS
LIN {X -41.5466,Y -71.5226,Z 84,A -125.515,B 24.9221,C -2.0378,E1 24.9185,E2 210.3729} C_DIS
LIN {X -44.3349,Y -69.8282,Z 84,A -127.7976,B 24.9219,C -2.0405,E1 24.9131,E2 212.6562} C_DIS
LIN {X -46.8791,Y -68.1463,Z 84,A -130.0248,B 24.9219,C -2.0407,E1 24.9079,E2 214.8903} C_DIS
LIN {X -49.8317,Y -66.0172,Z 84,A -132.8677,B 24.9223,C -2.0361,E1 24.9015,E2 217.7542} C_DIS
LIN {X -54.1185,Y -62.5522,Z 84,A -136.0162,B 24.9203,C -2.0617,E1 24.8949,E2 220.8537} C_DIS
LIN {X -56.7953,Y -60.1312,Z 84,A -139.3033,B 24.9216,C -2.0451,E1 24.888,E2 224.1937} C_DIS
LIN {X -59.8642,Y -57.0782,Z 84,A -141.865,B 24.9202,C -2.0634,E1 24.8831,E2 226.7229} C_DIS
LIN {X -62.9668,Y -53.6342,Z 84,A -145.4843,B 24.9205,C -2.0596,E1 24.8764,E2 230.3675} C_DIS
LIN {X -67.0738,Y -48.4018,Z 84,A -150.3527,B 24.9201,C -2.0637,E1 24.8682,E2 235.2494} C_DIS
LIN {X -69.1416,Y -45.3972,Z 84,A -152.1095,B 24.918,C -2.0907,E1 24.8655,E2 236.9507} C_DIS
LIN {X -70.9394,Y -42.5357,Z 84,A -154.9969,B 24.9187,C -2.0822,E1 24.8613,E2 239.8732} C_DIS
LIN {X -73.3684,Y -38.1926,Z 84,A -157.9056,B 24.9168,C -2.1058,E1 24.8575,E2 242.7408} C_DIS
LIN {X -74.6627,Y -35.5947,Z 84,A -160.966,B 24.9186,C -2.0837,E1 24.8537,E2 245.8705} C_DIS
LIN {X -76.4544,Y -31.5648,Z 84,A -163.1593,B 24.9161,C -2.115,E1 24.8514,E2 248.0013} C_DIS
LIN {X -77.6306,Y -28.5479,Z 84,A -165.3932,B 24.9156,C -2.1218,E1 24.8492,E2 250.2316} C_DIS
LIN {X -78.7285,Y -25.3627,Z 84,A -167.5724,B 24.9147,C -2.1328,E1 24.8472,E2 252.3971} C_DIS
LIN {X -79.5107,Y -22.7938,Z 84,A -170.5191,B 24.9165,C -2.11,E1 24.8449,E2 255.4153} C_DIS
LIN {X -80.6025,Y -18.5655,Z 84,A -172.1016,B 24.9127,C -2.1569,E1 24.844,E2 256.895} C_DIS
LIN {X -81.5184,Y -14.012,Z 84,A -175.9771,B 24.9133,C -2.1494,E1 24.8418,E2 260.8112} C_DIS
LIN {X -82.0431,Y -10.5065,Z 84,A -178.8449,B 24.9136,C -2.1464,E1 24.8407,E2 263.7034} C_DIS
LIN {X -82.5905,Y -4.5001,Z 84,A 177.9783,B 24.9104,C -2.1858,E1 24.84,E2 266.8053} C_DIS
LIN {X -82.6759,Y -2.4784,Z 84,A 176.0122,B 24.9112,C -2.1754,E1 24.8398,E2 268.808} C_DIS
LIN {X -82.6652,Y 2.8253,Z 84,A 172.6652,B 24.9096,C -2.1956,E1 24.8399,E2 272.1268} C_DIS
LIN {X -82.4754,Y 6.2735,Z 84,A 170.0585,B 24.9094,C -2.1977,E1 24.8403,E2 274.7444} C_DIS
LIN {X -82.2273,Y 8.9572,Z 84,A 168.0003,B 24.9094,C -2.1986,E1 24.8409,E2 276.8126} C_DIS
LIN {X -81.8201,Y 12.1284,Z 84,A 165.5077,B 24.9094,C -2.1985,E1 24.8419,E2 279.3204} C_DIS
LIN {X -80.5098,Y 18.967,Z 84,A 161.1372,B 24.9071,C -2.2255,E1 24.8443,E2 283.6522} C_DIS
LIN {X -79.2732,Y 23.6053,Z 84,A 157.3256,B 24.9073,C -2.2232,E1 24.8471,E2 287.4914} C_DIS
LIN {X -77.909,Y 27.7814,Z 84,A 154.7071,B 24.9056,C -2.2437,E1 24.8494,E2 290.076} C_DIS
LIN {X -76.7733,Y 30.7813,Z 84,A 152.1125,B 24.9058,C -2.2407,E1 24.8521,E2 292.6922} C_DIS
LIN {X -74.942,Y 35.0022,Z 84,A 149.5701,B 24.9036,C -2.2672,E1 24.8549,E2 295.1854} C_DIS
LIN {X -74.0473,Y 36.8573,Z 84,A 147.633,B 24.9044,C -2.2579,E1 24.8573,E2 297.155} C_DIS
LIN {X -71.51,Y 41.5684,Z 84,A 143.884,B 24.9035,C -2.2675,E1 24.8624,E2 300.901} C_DIS
LIN {X -68.856,Y 45.8304,Z 84,A 140.675,B 24.9021,C -2.2843,E1 24.8671,E2 304.086} C_DIS
LIN {X -66.1227,Y 49.6914,Z 84,A 137.3292,B 24.9015,C -2.2914,E1 24.8726,E2 307.4314} C_DIS
LIN {X -64.592,Y 51.6651,Z 84,A 134.6232,B 24.9033,C -2.2701,E1 24.8774,E2 310.2007} C_DIS
LIN {X -62.076,Y 54.6638,Z 84,A 132.1012,B 24.9023,C -2.2819,E1 24.882,E2 312.706} C_DIS
LIN {X -59.8838,Y 57.0567,Z 84,A 130.1592,B 24.9011,C -2.2956,E1 24.8857,E2 314.6239} C_DIS
LIN {X -56.6095,Y 60.306,Z 84,A 126.7293,B 24.9011,C -2.2968,E1 24.8926,E2 318.065} C_DIS
LIN {X -51.6854,Y 64.5759,Z 84,A 122.5999,B 24.8993,C -2.3171,E1 24.9013,E2 322.1619} C_DIS
LIN {X -49.1488,Y 66.5279,Z 84,A 119.5768,B 24.9007,C -2.3001,E1 24.9082,E2 325.2365} C_DIS
LIN {X -45.7761,Y 68.8918,Z 84,A 117.8627,B 24.8976,C -2.3364,E1 24.912,E2 326.8697} C_DIS
LIN {X -41.9814,Y 71.2672,Z 84,A 114.6414,B 24.8974,C -2.3388,E1 24.9197,E2 330.0954} C_DIS
LIN {X -39.524,Y 72.6588,Z 84,A 111.8549,B 24.8991,C -2.3195,E1 24.9266,E2 332.936} C_DIS
LIN {X -36.4347,Y 74.2568,Z 84,A 110.1026,B 24.8971,C -2.3413,E1 24.9309,E2 334.6409} C_DIS
LIN {X -33.8366,Y 75.4755,Z 84,A 108.1081,B 24.8969,C -2.3441,E1 24.9359,E2 336.6336} C_DIS
LIN {X -31.4107,Y 76.5171,Z 84,A 105.624,B 24.8983,C -2.3286,E1 24.9424,E2 339.1604} C_DIS
LIN {X -28.2538,Y 77.7378,Z 84,A 104.1912,B 24.8958,C -2.3569,E1 24.946,E2 340.5287} C_DIS
LIN {X -25.3389,Y 78.7363,Z 84,A 101.4271,B 24.8971,C -2.3418,E1 24.9535,E2 343.3337} C_DIS
LIN {X -21.6883,Y 79.819,Z 84,A 98.5854,B 24.8974,C -2.3389,E1 24.9611,E2 346.1869} C_DIS
LIN {X -17.4388,Y 80.854,Z 84,A 96.1097,B 24.8957,C -2.3572,E1 24.9678,E2 348.6223} C_DIS
LIN {X -14.1391,Y 81.4971,Z 84,A 93.4632,B 24.8964,C -2.35,E1 24.9751,E2 351.2888} C_DIS
LIN {X -9.4327,Y 82.1736,Z 84,A 90.4292,B 24.8955,C -2.3594,E1 24.9834,E2 354.3026} C_DIS
LIN {X -6.0231,Y 82.4946,Z 84,A 87.9644,B 24.8957,C -2.3578,E1 24.9903,E2 356.7723} C_DIS
LIN {X -1.5274,Y 82.6989,Z 84,A 84.4462,B 24.8966,C -2.3472,E1 25.0002,E2 360.3162} C_DIS
LIN {X 2.8023,Y 82.666,Z 84,A 81.9259,B 24.8954,C -2.3615,E1 25.0071,E2 362.8022} C_DIS
LIN {X 6.0991,Y 82.4893,Z 84,A 79.5646,B 24.8956,C -2.3593,E1 25.0137,E2 365.1677} C_DIS
LIN {X 10.115,Y 82.0931,Z 84,A 76.5724,B 24.8961,C -2.3531,E1 25.0221,E2 368.1726} C_DIS
LIN {X 13.4388,Y 81.6142,Z 84,A 74.5156,B 24.8955,C -2.3603,E1 25.0277,E2 370.2102} C_DIS
LIN {X 16.684,Y 81.0129,Z 84,A 71.8158,B 24.8966,C -2.3471,E1 25.0352,E2 372.938} C_DIS
LIN {X 20.3564,Y 80.1693,Z 84,A 69.3781,B 24.8963,C -2.3507,E1 25.0417,E2 375.3636} C_DIS
LIN {X 24.1676,Y 79.1043,Z 84,A 66.9142,B 24.8957,C -2.3571,E1 25.0483,E2 377.8083} C_DIS
LIN {X 27.8914,Y 77.8698,Z 84,A 63.8754,B 24.8968,C -2.3451,E1 25.0564,E2 380.8694} C_DIS
LIN {X 31.3131,Y 76.5568,Z 84,A 61.7948,B 24.8958,C -2.3565,E1 25.0617,E2 382.9184} C_DIS
LIN {X 35.8391,Y 74.5453,Z 84,A 58.2118,B 24.8966,C -2.3479,E1 25.0708,E2 386.5127} C_DIS
LIN {X 38.8266,Y 73.0345,Z 84,A 55.8546,B 24.8969,C -2.3438,E1 25.0767,E2 388.8733} C_DIS
LIN {X 42.5165,Y 70.9505,Z 84,A 52.9875,B 24.8971,C -2.3417,E1 25.0836,E2 391.7367} C_DIS
LIN {X 45.6877,Y 68.9501,Z 84,A 50.4576,B 24.8973,C -2.3397,E1 25.0895,E2 394.2629} C_DIS
LIN {X 50.5587,Y 65.462,Z 84,A 46.1847,B 24.8982,C -2.3288,E1 25.0992,E2 398.5466} C_DIS
LIN {X 53.2165,Y 63.3219,Z 84,A 42.9964,B 24.9009,C -2.2987,E1 25.1062,E2 401.7938} C_DIS
LIN {X 56.4633,Y 60.4435,Z 84,A 41.2339,B 24.898,C -2.3315,E1 25.1096,E2 403.4715} C_DIS
LIN {X 58.1739,Y 58.7983,Z 84,A 39.2666,B 24.8992,C -2.3179,E1 25.1136,E2 405.4629} C_DIS
LIN {X 62.1226,Y 54.6104,Z 84,A 35.3682,B 24.8997,C -2.3119,E1 25.121,E2 409.3583} C_DIS
LIN {X 63.7224,Y 52.7345,Z 84,A 33.5936,B 24.9002,C -2.3059,E1 25.1242,E2 411.1391} C_DIS
LIN {X 66.8248,Y 48.7433,Z 84,A 30.7201,B 24.8992,C -2.3176,E1 25.129,E2 413.9713} C_DIS
LIN {X 68.0348,Y 47.0398,Z 84,A 28.2023,B 24.9025,C -2.2797,E1 25.1332,E2 416.5664} C_DIS
LIN {X 70.0375,Y 44.0027,Z 84,A 25.5282,B 24.9035,C -2.2682,E1 25.1372,E2 419.254} C_DIS
LIN {X 71.8832,Y 40.919,Z 84,A 23.8312,B 24.9019,C -2.287,E1 25.1395,E2 420.898} C_DIS
LIN {X 73.0563,Y 38.7852,Z 84,A 22.0955,B 24.9024,C -2.2808,E1 25.1418,E2 422.6391} C_DIS
LIN {X 74.2648,Y 36.418,Z 84,A 20.1987,B 24.903,C -2.2739,E1 25.1442,E2 424.542} C_DIS
LIN {X 75.591,Y 33.5802,Z 84,A 17.4278,B 24.9052,C -2.2484,E1 25.1474,E2 427.3581} C_DIS
LIN {X 76.9116,Y 30.4317,Z 84,A 15.5926,B 24.9043,C -2.2587,E1 25.1493,E2 429.1589} C_DIS
LIN {X 78.2974,Y 26.664,Z 84,A 12.9607,B 24.9046,C -2.2554,E1 25.1517,E2 431.7839} C_DIS
LIN {X 80.2234,Y 20.146,Z 84,A 8.4591,B 24.9052,C -2.2479,E1 25.1552,E2 436.2773} C_DIS
LIN {X 80.8699,Y 17.3658,Z 84,A 6.4312,B 24.9059,C -2.2402,E1 25.1564,E2 438.3117} C_DIS
LIN {X 81.486,Y 14.2013,Z 84,A 3.9292,B 24.9072,C -2.2245,E1 25.1577,E2 440.8361} C_DIS
LIN {X 82.0413,Y 10.5202,Z 84,A 1.4347,B 24.9076,C -2.2192,E1 25.1587,E2 443.3285} C_DIS
LIN {X 82.3885,Y 7.3244,Z 84,A -0.716,B 24.908,C -2.2147,E1 25.1593,E2 445.4771} C_DIS
LIN {X 82.5817,Y 4.6594,Z 84,A -3.4913,B 24.911,C -2.1787,E1 25.1597,E2 448.3209} C_DIS
LIN {X 82.7131,Y 0.153,Z 84,A -5.367,B 24.9084,C -2.2094,E1 25.1598,E2 450.1128} C_DIS
LIN {X 82.6898,Y -2.0161,Z 84,A -7.6093,B 24.9108,C -2.1803,E1 25.1596,E2 452.4105} C_DIS
LIN {X 82.5335,Y -5.4475,Z 84,A -9.7902,B 24.9109,C -2.1792,E1 25.1593,E2 454.581} C_DIS
LIN {X 82.1769,Y -9.4049,Z 84,A -11.9997,B 24.9102,C -2.1883,E1 25.1587,E2 456.7561} C_DIS
LIN {X 81.494,Y -14.1567,Z 84,A -15.3495,B 24.9111,C -2.1768,E1 25.1573,E2 460.1133} C_DIS
LIN {X 80.9182,Y -17.1397,Z 84,A -17.7516,B 24.9125,C -2.1604,E1 25.1559,E2 462.5401} C_DIS
LIN {X 79.9204,Y -21.3131,Z 84,A -20.7694,B 24.9133,C -2.1495,E1 25.1539,E2 465.5662} C_DIS
LIN {X 78.1703,Y -27.0366,Z 84,A -24.7287,B 24.9139,C -2.1427,E1 25.1505,E2 469.519} C_DIS
LIN {X 75.9005,Y -32.8724,Z 84,A -29.0601,B 24.9149,C -2.1297,E1 25.146,E2 473.8571} C_DIS
LIN {X 73.6513,Y -37.6421,Z 84,A -32.2027,B 24.9145,C -2.1356,E1 25.1423,E2 476.969} C_DIS
LIN {X 71.7708,Y -41.1145,Z 84,A -35.0478,B 24.9154,C -2.124,E1 25.1385,E2 479.8265} C_DIS
LIN {X 68.9511,Y -45.6861,Z 84,A -39.0472,B 24.917,C -2.1044,E1 25.1325,E2 483.8521} C_DIS
LIN {X 67.2948,Y -48.0922,Z 84,A -41.9659,B 24.9196,C -2.07,E1 25.1277,E2 486.8378} C_DIS
LIN {X 64.6433,Y -51.6028,Z 84,A -43.8094,B 24.9172,C -2.1007,E1 25.1247,E2 488.6001} C_DIS
LIN {X 61.3442,Y -55.4843,Z 84,A -47.6002,B 24.9186,C -2.0831,E1 25.1177,E2 492.4154} C_DIS
LIN {X 58.4183,Y -58.555,Z 84,A -50.6484,B 24.9195,C -2.0724,E1 25.1117,E2 495.4757} C_DIS
LIN {X 55.5032,Y -61.3245,Z 84,A -53.6026,B 24.9204,C -2.0605,E1 25.1056,E2 498.4461} C_DIS
LIN {X 52.3491,Y -64.0401,Z 84,A -56.8573,B 24.9218,C -2.0423,E1 25.0986,E2 501.7313} C_DIS
LIN {X 49.4323,Y -66.3173,Z 84,A -58.4538,B 24.9198,C -2.0676,E1 25.0952,E2 503.2622} C_DIS
LIN {X 45.3688,Y -69.1604,Z 84,A -61.9204,B 24.9204,C -2.0597,E1 25.0872,E2 506.7356} C_DIS
LIN {X 42.723,Y -70.8256,Z 84,A -64.8166,B 24.9225,C -2.0326,E1 25.0802,E2 509.6868} C_DIS
LIN {X 39.935,Y -72.4351,Z 84,A -66.628,B 24.9218,C -2.0418,E1 25.0758,E2 511.4712} C_DIS
LIN {X 35.2494,Y -74.8269,Z 84,A -70.2006,B 24.9221,C -2.0381,E1 25.0669,E2 515.0428} C_DIS
LIN {X 31.5277,Y -76.4692,Z 84,A -73.0767,B 24.9226,C -2.0321,E1 25.0595,E2 517.9261} C_DIS
LIN {X 25.8608,Y -78.5672,Z 84,A -76.8857,B 24.9221,C -2.0384,E1 25.0496,E2 521.7125} C_DIS
LIN {X 23.2185,Y -79.3875,Z 84,A -79.5006,B 24.9239,C -2.0147,E1 25.0424,E2 524.3789} C_DIS
LIN {X 18.9809,Y -80.5066,Z 84,A -82.569,B 24.9242,C -2.0107,E1 25.0341,E2 527.4523} C_DIS
LIN {X 14.4273,Y -81.4453,Z 84,A -85.3135,B 24.9233,C -2.0225,E1 25.0266,E2 530.1655} C_DIS
LIN {X 11.1639,Y -81.9575,Z 84,A -88.2925,B 24.925,C -2.0001,E1 25.0183,E2 533.1951} C_DIS
LIN {X 7.4538,Y -82.3766,Z 84,A -90.1851,B 24.9235,C -2.0196,E1 25.0131,E2 535.0404} C_DIS
LIN {X 4.0567,Y -82.615,Z 84,A -92.6528,B 24.9238,C -2.0153,E1 25.0062,E2 537.5172} C_DIS
LIN {X 0.519,Y -82.7079,Z 84,A -94.0155,B 24.9214,C -2.0475,E1 25.0027,E2 538.8033} C_DIS
Enddeposition()
LIN {X 0.519,Y -82.7079,Z 84,A -94.0155,B 24.9214,C -2.0475,E1 25.0027,E2 538.8033} C_DIS
Startdeposition()
$VEL.CP = VEL_PRINT
LIN {X 1.1282,Y -81.7699,Z 84,A -93.0019,B 24.9187,C -2.0815,E1 25.0057,E2 537.7093} C_DIS
LIN {X 4.3397,Y -81.6618,Z 84,A -91.312,B 24.92,C -2.0653,E1 25.0103,E2 536.0583} C_DIS
LIN {X 7.5191,Y -81.4304,Z 84,A -88.3371,B 24.9182,C -2.0891,E1 25.0187,E2 533.0287} C_DIS
LIN {X 11.3152,Y -80.9905,Z 84,A -86.426,B 24.9199,C -2.0673,E1 25.0239,E2 531.1709} C_DIS
LIN {X 14.33,Y -80.5117,Z 84,A -84.3216,B 24.9199,C -2.0679,E1 25.0297,E2 529.0673} C_DIS
LIN {X 19.7661,Y -79.3531,Z 84,A -80.5531,B 24.9199,C -2.0675,E1 25.0399,E2 525.3047} C_DIS
LIN {X 24.7076,Y -77.9566,Z 84,A -76.7225,B 24.919,C -2.0787,E1 25.0503,E2 521.4542} C_DIS
LIN {X 27.4476,Y -77.034,Z 84,A -74.6859,B 24.9187,C -2.0816,E1 25.0556,E2 519.4147} C_DIS
LIN {X 31.7671,Y -75.3545,Z 84,A -71.3374,B 24.9181,C -2.0894,E1 25.0643,E2 516.0554} C_DIS
LIN {X 34.5112,Y -74.1379,Z 84,A -68.4697,B 24.916,C -2.1169,E1 25.0717,E2 513.1297} C_DIS
LIN {X 38.5927,Y -72.099,Z 84,A -66.4607,B 24.9185,C -2.0845,E1 25.0765,E2 511.2033} C_DIS
LIN {X 40.3133,Y -71.1495,Z 84,A -64.0785,B 24.9158,C -2.119,E1 25.0825,E2 508.7465} C_DIS
LIN {X 43.8024,Y -69.058,Z 84,A -62.1433,B 24.9177,C -2.095,E1 25.0869,E2 506.8741} C_DIS
LIN {X 45.6502,Y -67.8496,Z 84,A -60.4279,B 24.917,C -2.1034,E1 25.0909,E2 505.1446} C_DIS
LIN {X 48.3264,Y -65.9698,Z 84,A -58.0203,B 24.9164,C -2.1119,E1 25.0964,E2 502.7254} C_DIS
LIN {X 52.0322,Y -63.0888,Z 84,A -54.9926,B 24.9164,C -2.1106,E1 25.103,E2 499.7121} C_DIS
LIN {X 55.0866,Y -60.4393,Z 84,A -51.9439,B 24.9154,C -2.124,E1 25.1094,E2 496.6438} C_DIS
LIN {X 58.2013,Y -57.4462,Z 84,A -48.7701,B 24.9144,C -2.1361,E1 25.1157,E2 493.4549} C_DIS
LIN {X 60.907,Y -54.5692,Z 84,A -46.015,B 24.9139,C -2.1427,E1 25.1209,E2 490.6964} C_DIS
LIN {X 63.9531,Y -50.9664,Z 84,A -43.0575,B 24.9141,C -2.1399,E1 25.1261,E2 487.7591} C_DIS
LIN {X 65.9697,Y -48.3265,Z 84,A -40.5038,B 24.913,C -2.1536,E1 25.1304,E2 485.1854} C_DIS
LIN {X 67.5419,Y -46.1046,Z 84,A -38.3031,B 24.9118,C -2.1685,E1 25.1339,E2 482.9603} C_DIS
LIN {X 69.3244,Y -43.3772,Z 84,A -36.3543,B 24.9122,C -2.1639,E1 25.1368,E2 481.0321} C_DIS
LIN {X 72.7038,Y -37.4389,Z 84,A -32.1813,B 24.9127,C -2.1576,E1 25.1424,E2 476.8958} C_DIS
LIN {X 74.0469,Y -34.7067,Z 84,A -29.3668,B 24.9103,C -2.1863,E1 25.1458,E2 474.0286} C_DIS
LIN {X 76.0449,Y -30.0777,Z 84,A -25.8265,B 24.9094,C -2.1973,E1 25.1496,E2 470.4818} C_DIS
LIN {X 77.4897,Y -26.1305,Z 84,A -23.34,B 24.9099,C -2.1912,E1 25.1519,E2 468.0237} C_DIS
LIN {X 78.4127,Y -23.2144,Z 84,A -20.7378,B 24.9081,C -2.2131,E1 25.154,E2 465.3846} C_DIS
LIN {X 79.568,Y -18.8848,Z 84,A -18.015,B 24.9085,C -2.2091,E1 25.1559,E2 462.6869} C_DIS
LIN {X 80.2088,Y -15.9449,Z 84,A -15.9207,B 24.9079,C -2.2154,E1 25.157,E2 460.5901} C_DIS
LIN {X 81.1454,Y -10.1492,Z 84,A -12.0011,B 24.9074,C -2.222,E1 25.1587,E2 456.6778} C_DIS
LIN {X 81.5897,Y -5.5289,Z 84,A -8.3561,B 24.9054,C -2.2454,E1 25.1596,E2 452.9992} C_DIS
LIN {X 81.7646,Y -1.4199,Z 84,A -5.7567,B 24.9054,C -2.2453,E1 25.1598,E2 450.4156} C_DIS
LIN {X 81.7734,Y 0.8495,Z 84,A -3.505,B 24.9031,C -2.2723,E1 25.1598,E2 448.1135} C_DIS
LIN {X 81.6548,Y 4.4672,Z 84,A -1.674,B 24.9044,C -2.257,E1 25.1595,E2 446.3296} C_DIS
LIN {X 81.4086,Y 7.7554,Z 84,A 0.5269,B 24.9041,C -2.2606,E1 25.1589,E2 444.1331} C_DIS
LIN {X 81.0894,Y 10.5817,Z 84,A 2.5326,B 24.9036,C -2.2673,E1 25.1583,E2 442.1234} C_DIS
LIN {X 80.6407,Y 13.5843,Z 84,A 4.6869,B 24.9029,C -2.2749,E1 25.1573,E2 439.964} C_DIS
LIN {X 80.0783,Y 16.5811,Z 84,A 7.3457,B 24.9009,C -2.2987,E1 25.1558,E2 437.2644} C_DIS
LIN {X 79.3111,Y 19.9346,Z 84,A 10.0858,B 24.8993,C -2.3169,E1 25.154,E2 434.4971} C_DIS
LIN {X 78.1943,Y 23.9412,Z 84,A 12.2099,B 24.9008,C -2.2996,E1 25.1523,E2 432.4262} C_DIS
LIN {X 77.459,Y 26.2216,Z 84,A 14.0596,B 24.8999,C -2.3101,E1 25.1506,E2 430.5619} C_DIS
LIN {X 75.9507,Y 30.3176,Z 84,A 17.2491,B 24.8987,C -2.3233,E1 25.1474,E2 427.3591} C_DIS
LIN {X 74.3249,Y 34.1096,Z 84,A 19.6968,B 24.8993,C -2.317,E1 25.1446,E2 424.9395} C_DIS
LIN {X 73.0579,Y 36.7451,Z 84,A 21.7836,B 24.8987,C -2.3239,E1 25.142,E2 422.8476} C_DIS
LIN {X 71.6751,Y 39.3741,Z 84,A 23.6296,B 24.8988,C -2.3219,E1 25.1396,E2 421.016} C_DIS
LIN {X 69.5916,Y 42.9476,Z 84,A 26.4713,B 24.8983,C -2.3277,E1 25.1356,E2 418.1751} C_DIS
LIN {X 67.4057,Y 46.3048,Z 84,A 29.5052,B 24.8971,C -2.3422,E1 25.1309,E2 415.1222} C_DIS
LIN {X 65.9954,Y 48.2914,Z 84,A 32.1457,B 24.894,C -2.3766,E1 25.1264,E2 412.4131} C_DIS
LIN {X 63.1988,Y 51.8998,Z 84,A 34.3257,B 24.8963,C -2.3512,E1 25.1227,E2 410.3032} C_DIS
LIN {X 60.1951,Y 55.3535,Z 84,A 37.9707,B 24.8944,C -2.3724,E1 25.1159,E2 406.6243} C_DIS
LIN {X 57.159,Y 58.4849,Z 84,A 40.5476,B 24.8952,C -2.3636,E1 25.1108,E2 404.0792} C_DIS
LIN {X 51.8602,Y 63.2314,Z 84,A 45.4317,B 24.8946,C -2.3701,E1 25.1006,E2 399.199} C_DIS
LIN {X 48.5358,Y 65.8165,Z 84,A 48.8724,B 24.8927,C -2.3907,E1 25.0929,E2 395.7221} C_DIS
LIN {X 45.0497,Y 68.2494,Z 84,A 51.8124,B 24.8924,C -2.3943,E1 25.0861,E2 392.7834} C_DIS
LIN {X 42.16,Y 70.0723,Z 84,A 53.8371,B 24.8931,C -2.3864,E1 25.0813,E2 390.7838} C_DIS
LIN {X 39.3535,Y 71.6863,Z 84,A 56.152,B 24.8927,C -2.391,E1 25.0757,E2 388.4649} C_DIS
LIN {X 36.2406,Y 73.3081,Z 84,A 59.7003,B 24.8894,C -2.4278,E1 25.0666,E2 384.8387} C_DIS
LIN {X 31.674,Y 75.3938,Z 84,A 61.9739,B 24.8925,C -2.3933,E1 25.061,E2 382.6526} C_DIS
LIN {X 25.9103,Y 77.5639,Z 84,A 66.3956,B 24.8919,C -2.4004,E1 25.0494,E2 378.2232} C_DIS
LIN {X 23.1213,Y 78.4403,Z 84,A 68.9802,B 24.8903,C -2.4181,E1 25.0424,E2 375.601} C_DIS
LIN {X 19.9565,Y 79.3055,Z 84,A 70.5079,B 24.8922,C -2.3962,E1 25.0384,E2 374.1276} C_DIS
LIN {X 15.6398,Y 80.2676,Z 84,A 73.7959,B 24.8916,C -2.4034,E1 25.0294,E2 370.827} C_DIS
LIN {X 12.7245,Y 80.7812,Z 84,A 76.4137,B 24.8901,C -2.4203,E1 25.0221,E2 368.1717} C_DIS
LIN {X 7.8261,Y 81.4021,Z 84,A 79.3994,B 24.8913,C -2.4067,E1 25.0139,E2 365.2203} C_DIS
LIN {X 4.5691,Y 81.6491,Z 84,A 81.5846,B 24.8916,C -2.4037,E1 25.0078,E2 363.0431} C_DIS
LIN {X 2.1638,Y 81.749,Z 84,A 84.1114,B 24.8893,C -2.4282,E1 25.0006,E2 360.4585} C_DIS
LIN {X -1.7658,Y 81.7582,Z 84,A 86.5153,B 24.8903,C -2.4173,E1 24.9939,E2 358.0805} C_DIS
LIN {X -6.1294,Y 81.5477,Z 84,A 89.1389,B 24.8916,C -2.4033,E1 24.9867,E2 355.4892} C_DIS
LIN {X -9.2299,Y 81.2548,Z 84,A 91.8823,B 24.8902,C -2.4184,E1 24.979,E2 352.7082} C_DIS
LIN {X -12.4102,Y 80.8297,Z 84,A 93.5304,B 24.8919,C -2.3996,E1 24.9746,E2 351.1034} C_DIS
LIN {X -17.7477,Y 79.8284,Z 84,A 97.3735,B 24.8921,C -2.3976,E1 24.9641,E2 347.2609} C_DIS
LIN {X -22.7121,Y 78.5608,Z 84,A 101.0965,B 24.8921,C -2.3977,E1 24.954,E2 343.5319} C_DIS
LIN {X -27.1353,Y 77.1436,Z 84,A 104.1538,B 24.893,C -2.3883,E1 24.9459,E2 340.4913} C_DIS
LIN {X -30.9484,Y 75.6946,Z 84,A 107.8705,B 24.8911,C -2.4086,E1 24.9361,E2 336.7182} C_DIS
LIN {X -34.4507,Y 74.1661,Z 84,A 109.7452,B 24.8935,C -2.3821,E1 24.9315,E2 334.902} C_DIS
LIN {X -36.8127,Y 73.0233,Z 84,A 111.8691,B 24.8931,C -2.3871,E1 24.9262,E2 332.7607} C_DIS
LIN {X -40.5696,Y 71.0043,Z 84,A 114.7773,B 24.8937,C -2.3797,E1 24.9191,E2 329.8616} C_DIS
LIN {X -44.693,Y 68.4846,Z 84,A 117.7985,B 24.8952,C -2.3635,E1 24.912,E2 326.8697} C_DIS
LIN {X -49.4526,Y 65.1312,Z 84,A 121.9122,B 24.8958,C -2.3561,E1 24.9027,E2 322.7592} C_DIS
LIN {X -53.7342,Y 61.645,Z 84,A 125.5832,B 24.8971,C -2.3423,E1 24.8948,E2 319.1072} C_DIS
LIN {X -56.9075,Y 58.7285,Z 84,A 128.9016,B 24.897,C -2.3433,E1 24.888,E2 315.7729} C_DIS
LIN {X -58.3302,Y 57.3157,Z 84,A 131.4434,B 24.8945,C -2.3707,E1 24.8829,E2 313.1548} C_DIS
LIN {X -61.3697,Y 54.0493,Z 84,A 133.3471,B 24.8981,C -2.3299,E1 24.8795,E2 311.3401} C_DIS
LIN {X -64.7264,Y 49.9796,Z 84,A 136.8951,B 24.8993,C -2.3163,E1 24.8732,E2 307.808} C_DIS
LIN {X -67.9523,Y 45.4985,Z 84,A 141.6897,B 24.8981,C -2.3304,E1 24.8654,E2 302.9564} C_DIS
LIN {X -70.1829,Y 41.9761,Z 84,A 144.1161,B 24.9,C -2.309,E1 24.8619,E2 300.5687} C_DIS
LIN {X -71.8412,Y 39.0679,Z 84,A 146.8135,B 24.8997,C -2.3116,E1 24.8582,E2 297.8508} C_DIS
LIN {X -73.5933,Y 35.6589,Z 84,A 149.9222,B 24.8995,C -2.3149,E1 24.8544,E2 294.7174} C_DIS
LIN {X -75.0922,Y 32.3839,Z 84,A 151.9027,B 24.9014,C -2.2929,E1 24.8522,E2 292.7785} C_DIS
LIN {X -76.691,Y 28.3918,Z 84,A 154.7087,B 24.9026,C -2.2783,E1 24.8494,E2 289.9917} C_DIS
LIN {X -78.3929,Y 23.2812,Z 84,A 159.194,B 24.902,C -2.2854,E1 24.8455,E2 285.4638} C_DIS
LIN {X -79.2686,Y 20.0999,Z 84,A 161.0143,B 24.9037,C -2.2651,E1 24.8443,E2 283.6812} C_DIS
LIN {X -80.0072,Y 16.9241,Z 84,A 163.5897,B 24.9037,C -2.2656,E1 24.8428,E2 281.0896} C_DIS
LIN {X -80.9946,Y 11.2863,Z 84,A 167.2506,B 24.9056,C -2.2436,E1 24.8411,E2 277.4593} C_DIS
LIN {X -81.3798,Y 8.0617,Z 84,A 169.3927,B 24.9065,C -2.2329,E1 24.8405,E2 275.33} C_DIS
LIN {X -81.7086,Y 3.3455,Z 84,A 172.2997,B 24.9082,C -2.2117,E1 24.84,E2 272.456} C_DIS
LIN {X -81.758,Y -1.7765,Z 84,A 176.6042,B 24.9076,C -2.2189,E1 24.8399,E2 268.1085} C_DIS
LIN {X -81.572,Y -5.7791,Z 84,A 179.421,B 24.9084,C -2.2103,E1 24.8403,E2 265.2954} C_DIS
LIN {X -81.2468,Y -9.2922,Z 84,A -177.8052,B 24.9084,C -2.2105,E1 24.8411,E2 262.5044} C_DIS
LIN {X -80.693,Y -13.272,Z 84,A -175.116,B 24.9094,C -2.1983,E1 24.8423,E2 259.8282} C_DIS
LIN {X -79.6695,Y -18.4453,Z 84,A -170.8782,B 24.9091,C -2.2015,E1 24.8448,E2 255.558} C_DIS
LIN {X -78.7459,Y -22.0589,Z 84,A -168.9385,B 24.9112,C -2.1756,E1 24.8462,E2 253.6688} C_DIS
LIN {X -77.7415,Y -25.3724,Z 84,A -166.3318,B 24.9114,C -2.1732,E1 24.8484,E2 251.0528} C_DIS
LIN {X -76.4719,Y -28.9741,Z 84,A -163.8239,B 24.9124,C -2.1609,E1 24.8508,E2 248.56} C_DIS
LIN {X -74.5654,Y -33.5777,Z 84,A -159.7854,B 24.912,C -2.1657,E1 24.8553,E2 244.4879} C_DIS
LIN {X -72.6715,Y -37.5021,Z 84,A -157.3945,B 24.9142,C -2.1395,E1 24.8582,E2 242.1467} C_DIS
LIN {X -70.0905,Y -42.1301,Z 84,A -153.4143,B 24.9144,C -2.1367,E1 24.8638,E2 238.1523} C_DIS
LIN {X -68.4177,Y -44.7945,Z 84,A -150.7728,B 24.9139,C -2.143,E1 24.8678,E2 235.4825} C_DIS
LIN {X -64.9422,Y -49.6995,Z 84,A -147.0151,B 24.9157,C -2.1203,E1 24.8739,E2 231.7608} C_DIS
LIN {X -63.6022,Y -51.4026,Z 84,A -145.1564,B 24.9152,C -2.1261,E1 24.8772,E2 229.8797} C_DIS
LIN {X -59.5937,Y -56.0004,Z 84,A -141.3729,B 24.9171,C -2.103,E1 24.8842,E2 226.1341} C_DIS
LIN {X -56.0183,Y -59.5767,Z 84,A -137.2404,B 24.9163,C -2.112,E1 24.8925,E2 221.963} C_DIS
LIN {X -52.9815,Y -62.293,Z 84,A -133.7803,B 24.9154,C -2.1236,E1 24.9,E2 218.4618} C_DIS
LIN {X -49.3376,Y -65.2176,Z 84,A -131.4907,B 24.9181,C -2.09,E1 24.9049,E2 216.2438} C_DIS
LIN {X -47.455,Y -66.5994,Z 84,A -129.5943,B 24.9177,C -2.0946,E1 24.9092,E2 214.3299} C_DIS
LIN {X -42.8181,Y -69.6712,Z 84,A -125.9926,B 24.9188,C -2.0803,E1 24.9176,E2 210.7507} C_DIS
LIN {X -40.2071,Y -71.2109,Z 84,A -124.0854,B 24.9196,C -2.0712,E1 24.9222,E2 208.8595} C_DIS
LIN {X -35.4559,Y -73.6908,Z 84,A -120.0718,B 24.9194,C -2.0738,E1 24.9322,E2 204.8289} C_DIS
LIN {X -33.5366,Y -74.5839,Z 84,A -117.523,B 24.9171,C -2.103,E1 24.9389,E2 202.2045} C_DIS
LIN {X -29.1308,Y -76.4126,Z 84,A -115.2309,B 24.9197,C -2.0692,E1 24.9447,E2 199.9877} C_DIS
LIN {X -26.0344,Y -77.5221,Z 84,A -112.5283,B 24.919,C -2.0789,E1 24.9519,E2 197.257} C_DIS
LIN {X -22.4004,Y -78.6491,Z 84,A -109.5954,B 24.9185,C -2.085,E1 24.9598,E2 194.3048} C_DIS
LIN {X -18.9149,Y -79.5608,Z 84,A -107.635,B 24.9199,C -2.067,E1 24.965,E2 192.3845} C_DIS
LIN {X -15.6644,Y -80.2628,Z 84,A -104.9613,B 24.9192,C -2.0762,E1 24.9724,E2 189.6858} C_DIS
LIN {X -10.7207,Y -81.0714,Z 84,A -101.8914,B 24.9202,C -2.0623,E1 24.9808,E2 186.6464} C_DIS
LIN {X -6.9583,Y -81.4815,Z 84,A -98.9108,B 24.9195,C -2.0719,E1 24.9891,E2 183.6413} C_DIS
LIN {X -1.4889,Y -81.7633,Z 84,A -95.4381,B 24.9203,C -2.0613,E1 24.9988,E2 180.193} C_DIS
LIN {X 0.5119,Y -81.7746,Z 84,A -94.4233,B 24.9212,C -2.0501,E1 25.0015,E2 179.2051} C_DIS
Enddeposition()
LIN {X 0.5119,Y -81.7746,Z 84,A -94.4233,B 24.9212,C -2.0501,E1 25.0015,E2 179.2051} C_DIS
Startdeposition()
$VEL.CP = VEL_PRINT
LIN {X 0.1873,Y -80.8411,Z 84,A -95.3058,B 24.9214,C -2.0471,E1 24.999,E2 180.0945} C_DIS
LIN {X -5.2169,Y -80.6722,Z 84,A -99.2174,B 24.9216,C -2.0445,E1 24.9881,E2 184.0132} C_DIS
LIN {X -8.7185,Y -80.3698,Z 84,A -101.8216,B 24.9219,C -2.0414,E1 24.9808,E2 186.6261} C_DIS
LIN {X -12.3805,Y -79.8871,Z 84,A -104.895,B 24.9228,C -2.0291,E1 24.9723,E2 189.7313} C_DIS
LIN {X -15.9601,Y -79.2501,Z 84,A -106.8382,B 24.9213,C -2.048,E1 24.9671,E2 191.6317} C_DIS
LIN {X -20.89,Y -78.0952,Z 84,A -110.3307,B 24.921,C -2.0527,E1 24.9576,E2 195.118} C_DIS
LIN {X -25.0694,Y -76.8556,Z 84,A -113.4216,B 24.9208,C -2.0548,E1 24.9494,E2 198.2091} C_DIS
LIN {X -27.817,Y -75.9042,Z 84,A -115.6273,B 24.921,C -2.0526,E1 24.9435,E2 200.4245} C_DIS
LIN {X -33.0142,Y -73.7925,Z 84,A -119.5165,B 24.9205,C -2.059,E1 24.9335,E2 204.3073} C_DIS
LIN {X -38.0437,Y -71.3291,Z 84,A -123.8053,B 24.9208,C -2.0551,E1 24.9228,E2 208.6167} C_DIS
LIN {X -41.2726,Y -69.5113,Z 84,A -126.9773,B 24.9217,C -2.0441,E1 24.9151,E2 211.8247} C_DIS
LIN {X -44.7118,Y -67.3509,Z 84,A -128.8349,B 24.9192,C -2.0761,E1 24.9109,E2 213.6119} C_DIS
LIN {X -47.1346,Y -65.678,Z 84,A -131.0603,B 24.9192,C -2.0758,E1 24.9058,E2 215.8458} C_DIS
LIN {X -49.5823,Y -63.8507,Z 84,A -133.5478,B 24.9196,C -2.0709,E1 24.9002,E2 218.354} C_DIS
LIN {X -52.648,Y -61.3473,Z 84,A -136.1403,B 24.9187,C -2.0819,E1 24.8947,E2 220.9303} C_DIS
LIN {X -56.1286,Y -58.1791,Z 84,A -140.0957,B 24.9195,C -2.0722,E1 24.8866,E2 224.925} C_DIS
LIN {X -58.5979,Y -55.6928,Z 84,A -143.3532,B 24.9206,C -2.0574,E1 24.8802,E2 228.2319} C_DIS
LIN {X -62.3735,Y -51.4282,Z 84,A -146.0899,B 24.9173,C -2.1005,E1 24.8755,E2 230.8785} C_DIS
LIN {X -64.4731,Y -48.77,Z 84,A -148.3589,B 24.9165,C -2.1097,E1 24.8716,E2 233.1364} C_DIS
LIN {X -66.6148,Y -45.8022,Z 84,A -151.3168,B 24.9168,C -2.1066,E1 24.8668,E2 236.1161} C_DIS
LIN {X -68.5838,Y -42.7959,Z 84,A -153.4501,B 24.9154,C -2.1239,E1 24.8636,E2 238.2189} C_DIS
LIN {X -70.5842,Y -39.4093,Z 84,A -156.9087,B 24.9162,C -2.1139,E1 24.8588,E2 241.7193} C_DIS
LIN {X -73.3387,Y -34.0098,Z 84,A -161.1488,B 24.9151,C -2.1273,E1 24.8536,E2 245.9504} C_DIS
LIN {X -75.1858,Y -29.7042,Z 84,A -164.1016,B 24.9136,C -2.1462,E1 24.8505,E2 248.8746} C_DIS
LIN {X -76.2236,Y -26.9297,Z 84,A -166.1521,B 24.913,C -2.1536,E1 24.8485,E2 250.919} C_DIS
LIN {X -77.2259,Y -23.9036,Z 84,A -168.4736,B 24.9126,C -2.1587,E1 24.8465,E2 253.2416} C_DIS
LIN {X -77.999,Y -21.2462,Z 84,A -170.7841,B 24.9128,C -2.1557,E1 24.8448,E2 255.5726} C_DIS
LIN {X -78.821,Y -17.9592,Z 84,A -173.2491,B 24.9124,C -2.1614,E1 24.8432,E2 258.0385} C_DIS
LIN {X -79.8723,Y -12.4762,Z 84,A -177.1238,B 24.9112,C -2.1758,E1 24.8414,E2 261.9019} C_DIS
LIN {X -80.483,Y -7.598,Z 84,A 179.059,B 24.911,C -2.1784,E1 24.8402,E2 265.7357} C_DIS
LIN {X -80.7267,Y -4.295,Z 84,A 177.2204,B 24.9093,C -2.1986,E1 24.8399,E2 267.5371} C_DIS
LIN {X -80.839,Y 0.5119,Z 84,A 173.4042,B 24.9093,C -2.1992,E1 24.8399,E2 271.3749} C_DIS
LIN {X -80.3964,Y 8.4637,Z 84,A 168.1589,B 24.9069,C -2.2272,E1 24.8408,E2 276.5847} C_DIS
LIN {X -79.6846,Y 13.6238,Z 84,A 164.7355,B 24.9054,C -2.2458,E1 24.8422,E2 279.9842} C_DIS
LIN {X -79.0693,Y 16.8354,Z 84,A 162.0542,B 24.9055,C -2.2439,E1 24.8437,E2 282.6859} C_DIS
LIN {X -78.3665,Y 19.8493,Z 84,A 159.8665,B 24.905,C -2.2509,E1 24.8451,E2 284.8696} C_DIS
LIN {X -77.5125,Y 22.9571,Z 84,A 157.4733,B 24.9046,C -2.2553,E1 24.8469,E2 287.2662} C_DIS
LIN {X -76.0964,Y 27.2901,Z 84,A 154.5744,B 24.903,C -2.2737,E1 24.8495,E2 290.1378} C_DIS
LIN {X -75.0248,Y 30.1105,Z 84,A 151.9985,B 24.9034,C -2.2691,E1 24.8521,E2 292.7392} C_DIS
LIN {X -73.3495,Y 33.9865,Z 84,A 149.2123,B 24.9022,C -2.2833,E1 24.8553,E2 295.5067} C_DIS
LIN {X -72.2859,Y 36.195,Z 84,A 146.8554,B 24.9031,C -2.2727,E1 24.8583,E2 297.9016} C_DIS
LIN {X -70.7719,Y 39.0713,Z 84,A 145.1721,B 24.9012,C -2.2951,E1 24.8605,E2 299.5403} C_DIS
LIN {X -68.2589,Y 43.3124,Z 84,A 141.4911,B 24.9007,C -2.3002,E1 24.8658,E2 303.228} C_DIS
LIN {X -65.294,Y 47.6647,Z 84,A 137.4904,B 24.9004,C -2.3035,E1 24.8722,E2 307.2405} C_DIS
LIN {X -63.2859,Y 50.3008,Z 84,A 134.7666,B 24.9007,C -2.3,E1 24.877,E2 309.9853} C_DIS
LIN {X -60.9357,Y 53.1232,Z 84,A 133.3308,B 24.8975,C -2.3367,E1 24.8795,E2 311.3401} C_DIS
LIN {X -57.1145,Y 57.213,Z 84,A 129.1054,B 24.8973,C -2.3397,E1 24.8876,E2 315.577} C_DIS
LIN {X -53.3756,Y 60.7152,Z 84,A 125.5641,B 24.8963,C -2.3504,E1 24.8948,E2 319.1072} C_DIS
LIN {X -49.6657,Y 63.7864,Z 84,A 121.9639,B 24.8961,C -2.3528,E1 24.9026,E2 322.7151} C_DIS
LIN {X -47.8915,Y 65.128,Z 84,A 119.3312,B 24.8983,C -2.3284,E1 24.9086,E2 325.4153} C_DIS
LIN {X -44.4675,Y 67.512,Z 84,A 116.9748,B 24.8964,C -2.3498,E1 24.914,E2 327.7285} C_DIS
LIN {X -41.1672,Y 69.5736,Z 84,A 114.5472,B 24.8952,C -2.3636,E1 24.9197,E2 330.1307} C_DIS
LIN {X -36.6178,Y 72.0721,Z 84,A 110.7357,B 24.8949,C -2.3662,E1 24.9291,E2 333.9467} C_DIS
LIN {X -34.5399,Y 73.092,Z 84,A 108.1538,B 24.8969,C -2.3437,E1 24.9358,E2 336.5889} C_DIS
LIN {X -30.4861,Y 74.872,Z 84,A 105.7714,B 24.8948,C -2.3682,E1 24.9418,E2 338.9182} C_DIS
LIN {X -26.8784,Y 76.2416,Z 84,A 102.5819,B 24.8955,C -2.3594,E1 24.9503,E2 342.135} C_DIS
LIN {X -23.4942,Y 77.3525,Z 84,A 100.9106,B 24.8932,C -2.3855,E1 24.9546,E2 343.7473} C_DIS
LIN {X -19.2696,Y 78.5106,Z 84,A 97.69,B 24.8932,C -2.3855,E1 24.9633,E2 346.9729} C_DIS
LIN {X -16.3556,Y 79.1689,Z 84,A 95.079,B 24.8943,C -2.3736,E1 24.9705,E2 349.6151} C_DIS
LIN {X -12.9174,Y 79.8031,Z 84,A 92.1981,B 24.8951,C -2.3643,E1 24.9785,E2 352.5208} C_DIS
LIN {X -9.0271,Y 80.336,Z 84,A 90.1905,B 24.893,C -2.3873,E1 24.9839,E2 354.475} C_DIS
LIN {X -6.1465,Y 80.6072,Z 84,A 87.9289,B 24.8935,C -2.3824,E1 24.9902,E2 356.7494} C_DIS
LIN {X -1.8996,Y 80.8194,Z 84,A 84.0484,B 24.8956,C -2.3591,E1 25.0012,E2 360.6857} C_DIS
LIN {X 2.9278,Y 80.7889,Z 84,A 81.6445,B 24.893,C -2.388,E1 25.0077,E2 363.0205} C_DIS
LIN {X 5.2263,Y 80.6719,Z 84,A 79.6411,B 24.8939,C -2.3775,E1 25.0134,E2 365.0481} C_DIS
LIN {X 9.1386,Y 80.3229,Z 84,A 76.4933,B 24.8949,C -2.3667,E1 25.0222,E2 368.2193} C_DIS
LIN {X 13.0743,Y 79.7769,Z 84,A 74.4911,B 24.8929,C -2.3891,E1 25.0276,E2 370.1664} C_DIS
LIN {X 17.0897,Y 79.0138,Z 84,A 71.5025,B 24.8932,C -2.3852,E1 25.0358,E2 373.1606} C_DIS
LIN {X 22.1912,Y 77.7354,Z 84,A 67.9321,B 24.893,C -2.3875,E1 25.0454,E2 376.7201} C_DIS
LIN {X 24.967,Y 76.8887,Z 84,A 65.9196,B 24.893,C -2.3872,E1 25.0507,E2 378.7295} C_DIS
LIN {X 29.7497,Y 75.1679,Z 84,A 62.2924,B 24.8934,C -2.3832,E1 25.0602,E2 382.3586} C_DIS
LIN {X 32.1286,Y 74.1823,Z 84,A 60.2647,B 24.8941,C -2.3753,E1 25.0655,E2 384.4004} C_DIS
LIN {X 36.8533,Y 71.9518,Z 84,A 56.6341,B 24.8943,C -2.3729,E1 25.0746,E2 388.027} C_DIS
LIN {X 39.3417,Y 70.6219,Z 84,A 54.4213,B 24.8952,C -2.3638,E1 25.08,E2 390.2549} C_DIS
LIN {X 42.8998,Y 68.5189,Z 84,A 51.5532,B 24.8954,C -2.3613,E1 25.0869,E2 393.1199} C_DIS
LIN {X 45.5678,Y 66.7748,Z 84,A 49.1184,B 24.8962,C -2.3523,E1 25.0925,E2 395.5677} C_DIS
LIN {X 50.4797,Y 63.1445,Z 84,A 45.4128,B 24.8952,C -2.3636,E1 25.1007,E2 399.2332} C_DIS
LIN {X 52.2396,Y 61.6953,Z 84,A 43.3252,B 24.8967,C -2.3462,E1 25.1052,E2 401.354} C_DIS
LIN {X 56.1751,Y 58.1342,Z 84,A 39.9817,B 24.8963,C -2.3514,E1 25.112,E2 404.6715} C_DIS
LIN {X 59.2708,Y 54.9762,Z 84,A 36.2095,B 24.8986,C -2.325,E1 25.1194,E2 408.4899} C_DIS
LIN {X 61.8926,Y 52.0069,Z 84,A 32.7065,B 24.901,C -2.2972,E1 25.1258,E2 412.0425} C_DIS
LIN {X 65.1661,Y 47.8394,Z 84,A 30.2616,B 24.8983,C -2.3285,E1 25.1297,E2 414.4017} C_DIS
LIN {X 66.7748,Y 45.5678,Z 84,A 27.9323,B 24.8997,C -2.3124,E1 25.1335,E2 416.7576} C_DIS
LIN {X 69.4177,Y 41.431,Z 84,A 24.4467,B 24.9005,C -2.3032,E1 25.1386,E2 420.2474} C_DIS
LIN {X 71.4916,Y 37.7383,Z 84,A 22.1215,B 24.8993,C -2.3164,E1 25.1416,E2 422.5292} C_DIS
LIN {X 72.7503,Y 35.2517,Z 84,A 19.8147,B 24.9007,C -2.3004,E1 25.1445,E2 424.8613} C_DIS
LIN {X 74.2138,Y 32.0562,Z 84,A 17.2264,B 24.9016,C -2.2903,E1 25.1475,E2 427.4595} C_DIS
LIN {X 76.1648,Y 27.0973,Z 84,A 13.5792,B 24.9022,C -2.2834,E1 25.1511,E2 431.1026} C_DIS
LIN {X 77.1214,Y 24.2405,Z 84,A 11.0738,B 24.9037,C -2.2654,E1 25.1533,E2 433.6364} C_DIS
LIN {X 78.4355,Y 19.5775,Z 84,A 7.3174,B 24.9055,C -2.2448,E1 25.1559,E2 437.4199} C_DIS
LIN {X 79.29,Y 15.7655,Z 84,A 5.2982,B 24.9042,C -2.26,E1 25.157,E2 439.3914} C_DIS
LIN {X 79.8314,Y 12.7404,Z 84,A 3.0867,B 24.9048,C -2.2522,E1 25.1581,E2 441.6084} C_DIS
LIN {X 80.3106,Y 9.2443,Z 84,A 0.6415,B 24.9054,C -2.2461,E1 25.1589,E2 444.0534} C_DIS
LIN {X 80.6263,Y 5.901,Z 84,A -1.7314,B 24.906,C -2.2388,E1 25.1595,E2 446.4296} C_DIS
LIN {X 80.8264,Y 1.5189,Z 84,A -4.774,B 24.9066,C -2.2311,E1 25.1598,E2 449.4723} C_DIS
LIN {X 80.8245,Y -1.6228,Z 84,A -6.8948,B 24.9069,C -2.2274,E1 25.1598,E2 451.5893} C_DIS
LIN {X 80.7212,Y -4.3952,Z 84,A -8.9136,B 24.9076,C -2.2194,E1 25.1595,E2 453.6149} C_DIS
LIN {X 80.3466,Y -8.9363,Z 84,A -12.0296,B 24.9082,C -2.2127,E1 25.1587,E2 456.7282} C_DIS
LIN {X 79.7865,Y -13.0149,Z 84,A -14.9718,B 24.909,C -2.2026,E1 25.1575,E2 459.6769} C_DIS
LIN {X 79.1225,Y -16.5817,Z 84,A -17.4536,B 24.9094,C -2.1973,E1 25.1562,E2 462.1566} C_DIS
LIN {X 78.4243,Y -19.6228,Z 84,A -20.223,B 24.9115,C -2.1725,E1 25.1543,E2 464.9687} C_DIS
LIN {X 77.5278,Y -22.9056,Z 84,A -22.4574,B 24.9116,C -2.1706,E1 25.1526,E2 467.1947} C_DIS
LIN {X 76.27,Y -26.7974,Z 84,A -24.8178,B 24.911,C -2.1789,E1 25.1505,E2 469.5222} C_DIS
LIN {X 74.3676,Y -31.6983,Z 84,A -29.4119,B 24.9141,C -2.1398,E1 25.1457,E2 474.1831} C_DIS
LIN {X 72.9161,Y -34.9066,Z 84,A -31.4007,B 24.9134,C -2.1485,E1 25.1433,E2 476.1408} C_DIS
LIN {X 69.7225,Y -40.9153,Z 84,A -35.7721,B 24.9134,C -2.1489,E1 25.1375,E2 480.4884} C_DIS
LIN {X 66.9732,Y -45.2749,Z 84,A -39.3958,B 24.9141,C -2.1395,E1 25.1321,E2 484.1159} C_DIS
LIN {X 64.628,Y -48.5638,Z 84,A -42.7178,B 24.9159,C -2.1172,E1 25.1266,E2 487.4746} C_DIS
LIN {X 61.2175,Y -52.7996,Z 84,A -46.4039,B 24.9163,C -2.1124,E1 25.12,E2 491.155} C_DIS
LIN {X 59.6934,Y -54.5156,Z 84,A -48.0209,B 24.9166,C -2.1086,E1 25.117,E2 492.7738} C_DIS
LIN {X 57.1973,Y -57.1297,Z 84,A -50.5717,B 24.9171,C -2.1027,E1 25.112,E2 495.3277} C_DIS
LIN {X 53.3369,Y -60.749,Z 84,A -54.2589,B 24.9176,C -2.096,E1 25.1045,E2 499.0158} C_DIS
LIN {X 50.2156,Y -63.3532,Z 84,A -57.6312,B 24.9193,C -2.0745,E1 25.097,E2 502.4263} C_DIS
LIN {X 45.9352,Y -66.5225,Z 84,A -61.024,B 24.919,C -2.0785,E1 25.0894,E2 505.7976} C_DIS
LIN {X 43.0524,Y -68.4235,Z 84,A -64.3638,B 24.9215,C -2.0466,E1 25.0814,E2 509.2022} C_DIS
LIN {X 38.9127,Y -70.8604,Z 84,A -66.6616,B 24.9193,C -2.0743,E1 25.0759,E2 511.4276} C_DIS
LIN {X 33.773,Y -73.4489,Z 84,A -70.5513,B 24.9193,C -2.0735,E1 25.0662,E2 515.3088} C_DIS
LIN {X 32.0075,Y -74.2349,Z 84,A -72.6295,B 24.9212,C -2.0499,E1 25.0608,E2 517.4378} C_DIS
LIN {X 27.1144,Y -76.1588,Z 84,A -75.8879,B 24.9205,C -2.0591,E1 25.0523,E2 520.6676} C_DIS
LIN {X 24.2788,Y -77.1096,Z 84,A -78.6822,B 24.9222,C -2.0364,E1 25.0448,E2 523.5106} C_DIS
LIN {X 20.6749,Y -78.1526,Z 84,A -80.3554,B 24.9202,C -2.063,E1 25.0404,E2 525.118} C_DIS
LIN {X 18.2213,Y -78.7604,Z 84,A -82.8669,B 24.922,C -2.0398,E1 25.0335,E2 527.6809} C_DIS
LIN {X 13.7469,Y -79.6644,Z 84,A -85.9307,B 24.9218,C -2.0422,E1 25.0251,E2 530.7354} C_DIS
LIN {X 10.8354,Y -80.1125,Z 84,A -88.3378,B 24.9226,C -2.0315,E1 25.0184,E2 533.1661} C_DIS
LIN {X 7.4489,Y -80.4968,Z 84,A -90.0887,B 24.9212,C -2.0497,E1 25.0136,E2 534.8727} C_DIS
LIN {X 4.5805,Y -80.7109,Z 84,A -92.5183,B 24.9222,C -2.0373,E1 25.0068,E2 537.3305} C_DIS
LIN {X 0.5002,Y -80.8371,Z 84,A -94.1888,B 24.9195,C -2.0724,E1 25.0023,E2 538.9176} C_DIS
Enddeposition()
LIN {X 0.5002,Y -80.8371,Z 84,A -94.1888,B 24.9195,C -2.0724,E1 25.0023,E2 538.9176} C_DIS
Startdeposition()
$VEL.CP = VEL_PRINT
LIN {X 1.3491,Y -79.8933,Z 84,A -93.4934,B 24.918,C -2.0912,E1 25.0044,E2 538.1775} C_DIS
LIN {X 4.855,Y -79.7582,Z 84,A -91.1111,B 24.9182,C -2.0882,E1 25.011,E2 535.8032} C_DIS
LIN {X 7.4711,Y -79.5546,Z 84,A -88.6157,B 24.9167,C -2.1075,E1 25.0181,E2 533.2636} C_DIS
LIN {X 12.4396,Y -78.9307,Z 84,A -85.0484,B 24.9166,C -2.1092,E1 25.0279,E2 529.6954} C_DIS
LIN {X 17.6568,Y -77.93,Z 84,A -81.461,B 24.9168,C -2.1058,E1 25.0377,E2 526.1205} C_DIS
LIN {X 21.6536,Y -76.9147,Z 84,A -78.3954,B 24.9163,C -2.1122,E1 25.046,E2 523.0446} C_DIS
LIN {X 24.6727,Y -76,Z 84,A -76.3796,B 24.9167,C -2.1074,E1 25.0513,E2 521.0439} C_DIS
LIN {X 27.459,Y -75.0383,Z 84,A -74.2696,B 24.9165,C -2.11,E1 25.0569,E2 518.932} C_DIS
LIN {X 30.9183,Y -73.6804,Z 84,A -71.7393,B 24.9165,C -2.1097,E1 25.0634,E2 516.4083} C_DIS
LIN {X 32.7018,Y -72.9064,Z 84,A -70.0084,B 24.9155,C -2.1221,E1 25.0679,E2 514.6522} C_DIS
LIN {X 37.4115,Y -70.6056,Z 84,A -66.4453,B 24.9155,C -2.1222,E1 25.0767,E2 511.0985} C_DIS
LIN {X 39.5843,Y -69.411,Z 84,A -64.1966,B 24.9141,C -2.14,E1 25.0823,E2 508.8144} C_DIS
LIN {X 42.3849,Y -67.7367,Z 84,A -62.8594,B 24.9162,C -2.1132,E1 25.0853,E2 507.5449} C_DIS
LIN {X 44.3809,Y -66.4477,Z 84,A -60.4927,B 24.9143,C -2.1371,E1 25.0909,E2 505.1294} C_DIS
LIN {X 47.0845,Y -64.5586,Z 84,A -58.4178,B 24.9147,C -2.1329,E1 25.0956,E2 503.0719} C_DIS
LIN {X 51.227,Y -61.3235,Z 84,A -54.6421,B 24.914,C -2.1413,E1 25.1039,E2 499.2905} C_DIS
LIN {X 53.6216,Y -59.2417,Z 84,A -52.1156,B 24.9129,C -2.1544,E1 25.1092,E2 496.7431} C_DIS
LIN {X 56.9532,Y -56.0452,Z 84,A -48.6255,B 24.9118,C -2.1681,E1 25.1161,E2 493.2353} C_DIS
LIN {X 59.3074,Y -53.5489,Z 84,A -46.6201,B 24.9125,C -2.1597,E1 25.1199,E2 491.2584} C_DIS
LIN {X 61.5389,Y -50.9678,Z 84,A -44.1785,B 24.912,C -2.1659,E1 25.1243,E2 488.8134} C_DIS
LIN {X 63.2684,Y -48.8042,Z 84,A -41.3172,B 24.9093,C -2.1993,E1 25.1293,E2 485.8868} C_DIS
LIN {X 65.8143,Y -45.3138,Z 84,A -39.3317,B 24.9115,C -2.172,E1 25.1323,E2 483.9755} C_DIS
LIN {X 68.0739,Y -41.8431,Z 84,A -36.1365,B 24.9102,C -2.1875,E1 25.1372,E2 480.7597} C_DIS
LIN {X 70.1528,Y -38.2538,Z 84,A -32.9384,B 24.9089,C -2.2033,E1 25.1415,E2 477.5408} C_DIS
LIN {X 71.7801,Y -35.1075,Z 84,A -30.5943,B 24.9089,C -2.2045,E1 25.1445,E2 475.2065} C_DIS
LIN {X 73.4456,Y -31.4757,Z 84,A -27.8513,B 24.9085,C -2.2092,E1 25.1476,E2 472.4674} C_DIS
LIN {X 75.0373,Y -27.4619,Z 84,A -25.2567,B 24.909,C -2.2025,E1 25.1502,E2 469.9028} C_DIS
LIN {X 76.1692,Y -24.1499,Z 84,A -22.1403,B 24.9067,C -2.2298,E1 25.153,E2 466.7397} C_DIS
LIN {X 77.4032,Y -19.8363,Z 84,A -19.2685,B 24.9068,C -2.2287,E1 25.1551,E2 463.8869} C_DIS
LIN {X 77.9044,Y -17.7677,Z 84,A -17.5698,B 24.9059,C -2.2391,E1 25.1562,E2 462.1735} C_DIS
LIN {X 78.6398,Y -14.1604,Z 84,A -15.1761,B 24.9059,C -2.2395,E1 25.1574,E2 459.7927} C_DIS
LIN {X 79.29,Y -9.8979,Z 84,A -12.0665,B 24.905,C -2.2499,E1 25.1587,E2 456.6769} C_DIS
LIN {X 79.6386,Y -6.5155,Z 84,A -9.5591,B 24.9042,C -2.26,E1 25.1594,E2 454.1607} C_DIS
LIN {X 79.8206,Y -3.6688,Z 84,A -7.4936,B 24.9036,C -2.2671,E1 25.1597,E2 452.0906} C_DIS
LIN {X 79.9021,Y -0.6746,Z 84,A -5.285,B 24.9028,C -2.276,E1 25.1597,E2 449.8743} C_DIS
Enddeposition()
END
